OpModVal(
    bEn := TRUE,
    nSel := eOpMode,
    nEn01 := E_BA_AC_OpMod01.eOff,
    bVal01 := arrOpModVal[E_BA_AC_OpMod01.eOff],
    nEn02 := E_BA_AC_OpMod01.eOn,
    bVal02 := arrOpModVal[E_BA_AC_OpMod01.eOn],
    nEn03 := E_BA_AC_OpMod01.eEmergency,
    bVal03 := arrOpModVal[E_BA_AC_OpMod01.eEmergency],
    nEn04 := E_BA_AC_OpMod01.eFrost,
    bVal04 := arrOpModVal[E_BA_AC_OpMod01.eFrost],
    nEn05 := E_BA_AC_OpMod01.eSmokeExtractionProgram,
    bVal05 := arrOpModVal[E_BA_AC_OpMod01.eSmokeExtractionProgram],
    nEn06 := E_BA_AC_OpMod01.eSmokeExtractionSupplyAir,
    bVal06 := arrOpModVal[E_BA_AC_OpMod01.eSmokeExtractionSupplyAir],
    nEn07 := E_BA_AC_OpMod01.eSmokeExtractionExhaustAir,
    bVal07 := arrOpModVal[E_BA_AC_OpMod01.eSmokeExtractionExhaustAir],
    nEn08 := E_BA_AC_OpMod01.eFire,
    bVal08 := arrOpModVal[E_BA_AC_OpMod01.eFire],
    nEn09 := E_BA_AC_OpMod01.eNightCooling,
    bVal09 := arrOpModVal[E_BA_AC_OpMod01.eNightCooling],
    nEn10 := E_BA_AC_OpMod01.eCoolDownProtection,
    bVal10 := arrOpModVal[E_BA_AC_OpMod01.eCoolDownProtection],
    nEn11 := E_BA_AC_OpMod01.eOverHeatingProtection,
    bVal11 := arrOpModVal[E_BA_AC_OpMod01.eOverHeatingProtection],
    nEn12 := E_BA_AC_OpMod01.eAlarm,
    bVal12 := arrOpModVal[E_BA_AC_OpMod01.eAlarm],
    nEn13 := E_BA_AC_OpMod01.eForcedVentilation,
    bVal13 := arrOpModVal[E_BA_AC_OpMod01.eForcedVentilation],
    nEn14 := E_BA_AC_OpMod01.eCentralSwitchOff,
    bVal14 := arrOpModVal[E_BA_AC_OpMod01.eCentralSwitchOff],
    nEn15 := E_BA_AC_OpMod01.eCustomer01,
    bVal15 := arrOpModVal[E_BA_AC_OpMod01.eCustomer01],
    nEn16 := E_BA_AC_OpMod01.eCustomer02,
    bVal16 := arrOpModVal[E_BA_AC_OpMod01.eCustomer02],
    bReplVal := FALSE); // FB_BA_MMUX_B16
bVal := OpModVal.bVal;
_w1 := TO_UDINT(MAX(fDlyOn, 0));
DelayOn(
    bEn := TRUE,
    nSel := eOpMode,
    nEn01 := E_BA_AC_OpMod01.eOff,
    bVal01 := arrIgnoreDelayOnVal[E_BA_AC_OpMod01.eOff],
    nEn02 := E_BA_AC_OpMod01.eOn,
    bVal02 := arrIgnoreDelayOnVal[E_BA_AC_OpMod01.eOn],
    nEn03 := E_BA_AC_OpMod01.eEmergency,
    bVal03 := arrIgnoreDelayOnVal[E_BA_AC_OpMod01.eEmergency],
    nEn04 := E_BA_AC_OpMod01.eFrost,
    bVal04 := arrIgnoreDelayOnVal[E_BA_AC_OpMod01.eFrost],
    nEn05 := E_BA_AC_OpMod01.eSmokeExtractionProgram,
    bVal05 := arrIgnoreDelayOnVal[E_BA_AC_OpMod01.eSmokeExtractionProgram],
    nEn06 := E_BA_AC_OpMod01.eSmokeExtractionSupplyAir,
    bVal06 := arrIgnoreDelayOnVal[E_BA_AC_OpMod01.eSmokeExtractionSupplyAir],
    nEn07 := E_BA_AC_OpMod01.eSmokeExtractionExhaustAir,
    bVal07 := arrIgnoreDelayOnVal[E_BA_AC_OpMod01.eSmokeExtractionExhaustAir],
    nEn08 := E_BA_AC_OpMod01.eFire,
    bVal08 := arrIgnoreDelayOnVal[E_BA_AC_OpMod01.eFire],
    nEn09 := E_BA_AC_OpMod01.eNightCooling,
    bVal09 := arrIgnoreDelayOnVal[E_BA_AC_OpMod01.eNightCooling],
    nEn10 := E_BA_AC_OpMod01.eCoolDownProtection,
    bVal10 := arrIgnoreDelayOnVal[E_BA_AC_OpMod01.eCoolDownProtection],
    nEn11 := E_BA_AC_OpMod01.eOverHeatingProtection,
    bVal11 := arrIgnoreDelayOnVal[E_BA_AC_OpMod01.eOverHeatingProtection],
    nEn12 := E_BA_AC_OpMod01.eAlarm,
    bVal12 := arrIgnoreDelayOnVal[E_BA_AC_OpMod01.eAlarm],
    nEn13 := E_BA_AC_OpMod01.eForcedVentilation,
    bVal13 := arrIgnoreDelayOnVal[E_BA_AC_OpMod01.eForcedVentilation],
    nEn14 := E_BA_AC_OpMod01.eCentralSwitchOff,
    bVal14 := arrIgnoreDelayOnVal[E_BA_AC_OpMod01.eCentralSwitchOff],
    nEn15 := E_BA_AC_OpMod01.eCustomer01,
    bVal15 := arrIgnoreDelayOnVal[E_BA_AC_OpMod01.eCustomer01],
    nEn16 := E_BA_AC_OpMod01.eCustomer02,
    bVal16 := arrIgnoreDelayOnVal[E_BA_AC_OpMod01.eCustomer02],
    bReplVal := FALSE); // FB_BA_MMUX_B16
nDelayOn := SEL(DelayOn.bVal, _w1, 0);
_w2 := TO_UDINT(MAX(fDlyOff, 0));
DelayOff(
    bEn := TRUE,
    nSel := eOpMode,
    nEn01 := E_BA_AC_OpMod01.eOff,
    bVal01 := arrIgnoreDelayOffVal[E_BA_AC_OpMod01.eOff],
    nEn02 := E_BA_AC_OpMod01.eOn,
    bVal02 := arrIgnoreDelayOffVal[E_BA_AC_OpMod01.eOn],
    nEn03 := E_BA_AC_OpMod01.eEmergency,
    bVal03 := arrIgnoreDelayOffVal[E_BA_AC_OpMod01.eEmergency],
    nEn04 := E_BA_AC_OpMod01.eFrost,
    bVal04 := arrIgnoreDelayOffVal[E_BA_AC_OpMod01.eFrost],
    nEn05 := E_BA_AC_OpMod01.eSmokeExtractionProgram,
    bVal05 := arrIgnoreDelayOffVal[E_BA_AC_OpMod01.eSmokeExtractionProgram],
    nEn06 := E_BA_AC_OpMod01.eSmokeExtractionSupplyAir,
    bVal06 := arrIgnoreDelayOffVal[E_BA_AC_OpMod01.eSmokeExtractionSupplyAir],
    nEn07 := E_BA_AC_OpMod01.eSmokeExtractionExhaustAir,
    bVal07 := arrIgnoreDelayOffVal[E_BA_AC_OpMod01.eSmokeExtractionExhaustAir],
    nEn08 := E_BA_AC_OpMod01.eFire,
    bVal08 := arrIgnoreDelayOffVal[E_BA_AC_OpMod01.eFire],
    nEn09 := E_BA_AC_OpMod01.eNightCooling,
    bVal09 := arrIgnoreDelayOffVal[E_BA_AC_OpMod01.eNightCooling],
    nEn10 := E_BA_AC_OpMod01.eCoolDownProtection,
    bVal10 := arrIgnoreDelayOffVal[E_BA_AC_OpMod01.eCoolDownProtection],
    nEn11 := E_BA_AC_OpMod01.eOverHeatingProtection,
    bVal11 := arrIgnoreDelayOffVal[E_BA_AC_OpMod01.eOverHeatingProtection],
    nEn12 := E_BA_AC_OpMod01.eAlarm,
    bVal12 := arrIgnoreDelayOffVal[E_BA_AC_OpMod01.eAlarm],
    nEn13 := E_BA_AC_OpMod01.eForcedVentilation,
    bVal13 := arrIgnoreDelayOffVal[E_BA_AC_OpMod01.eForcedVentilation],
    nEn14 := E_BA_AC_OpMod01.eCentralSwitchOff,
    bVal14 := arrIgnoreDelayOffVal[E_BA_AC_OpMod01.eCentralSwitchOff],
    nEn15 := E_BA_AC_OpMod01.eCustomer01,
    bVal15 := arrIgnoreDelayOffVal[E_BA_AC_OpMod01.eCustomer01],
    nEn16 := E_BA_AC_OpMod01.eCustomer02,
    bVal16 := arrIgnoreDelayOffVal[E_BA_AC_OpMod01.eCustomer02],
    bReplVal := FALSE); // FB_BA_MMUX_B16
nDelayOff := SEL(DelayOff.bVal, _w2, 0);
IgnoreFdb(
    bEn := TRUE,
    nSel := eOpMode,
    nEn01 := E_BA_AC_OpMod01.eOff,
    bVal01 := arrIgnoreFdbVal[E_BA_AC_OpMod01.eOff],
    nEn02 := E_BA_AC_OpMod01.eOn,
    bVal02 := arrIgnoreFdbVal[E_BA_AC_OpMod01.eOn],
    nEn03 := E_BA_AC_OpMod01.eEmergency,
    bVal03 := arrIgnoreFdbVal[E_BA_AC_OpMod01.eEmergency],
    nEn04 := E_BA_AC_OpMod01.eFrost,
    bVal04 := arrIgnoreFdbVal[E_BA_AC_OpMod01.eFrost],
    nEn05 := E_BA_AC_OpMod01.eSmokeExtractionProgram,
    bVal05 := arrIgnoreFdbVal[E_BA_AC_OpMod01.eSmokeExtractionProgram],
    nEn06 := E_BA_AC_OpMod01.eSmokeExtractionSupplyAir,
    bVal06 := arrIgnoreFdbVal[E_BA_AC_OpMod01.eSmokeExtractionSupplyAir],
    nEn07 := E_BA_AC_OpMod01.eSmokeExtractionExhaustAir,
    bVal07 := arrIgnoreFdbVal[E_BA_AC_OpMod01.eSmokeExtractionExhaustAir],
    nEn08 := E_BA_AC_OpMod01.eFire,
    bVal08 := arrIgnoreFdbVal[E_BA_AC_OpMod01.eFire],
    nEn09 := E_BA_AC_OpMod01.eNightCooling,
    bVal09 := arrIgnoreFdbVal[E_BA_AC_OpMod01.eNightCooling],
    nEn10 := E_BA_AC_OpMod01.eCoolDownProtection,
    bVal10 := arrIgnoreFdbVal[E_BA_AC_OpMod01.eCoolDownProtection],
    nEn11 := E_BA_AC_OpMod01.eOverHeatingProtection,
    bVal11 := arrIgnoreFdbVal[E_BA_AC_OpMod01.eOverHeatingProtection],
    nEn12 := E_BA_AC_OpMod01.eAlarm,
    bVal12 := arrIgnoreFdbVal[E_BA_AC_OpMod01.eAlarm],
    nEn13 := E_BA_AC_OpMod01.eForcedVentilation,
    bVal13 := arrIgnoreFdbVal[E_BA_AC_OpMod01.eForcedVentilation],
    nEn14 := E_BA_AC_OpMod01.eCentralSwitchOff,
    bVal14 := arrIgnoreFdbVal[E_BA_AC_OpMod01.eCentralSwitchOff],
    nEn15 := E_BA_AC_OpMod01.eCustomer01,
    bVal15 := arrIgnoreFdbVal[E_BA_AC_OpMod01.eCustomer01],
    nEn16 := E_BA_AC_OpMod01.eCustomer02,
    bVal16 := arrIgnoreFdbVal[E_BA_AC_OpMod01.eCustomer02],
    bReplVal := FALSE); // FB_BA_MMUX_B16
_bFdb := SEL(IgnoreFdb.bVal, bFdb, TRUE);

END_FUNCTION_BLOCK

// ---- Templates/POUs/Trade/AirConditioning/General/FB_BA_AC_OpModAggMdlt.TcPOU
{region '#Template'}
	{attribute 'Version' := '5.1.0.0'}
	{attribute 'Tags' := '"LCID": "1031", "Text": "AC, Allgemein, AHU, Betriebsart"'}
	{attribute 'Tags' := '"LCID": "1033", "Text": "AC, General, AHU, Operating mode"'}
	{attribute 'Using' := '"Type": "Template", "URI": "E_BA_AC_OpMod01"'}
	{attribute 'Description' := '"LCID": "1031", "Text": "Betriebsart"'}
	{attribute 'Description' := '"LCID": "1033", "Text": "Operating mode"'}
{endregion}

FUNCTION_BLOCK FB_BA_AC_OpModAggMdlt
VAR_INPUT
	stPriorityEn				: ST_BA_PriorityEn;	
	eOpMode					: E_BA_AC_OpMod01;
	bFdb					: BOOL;
	fDlyOn					: REAL;	
	fDlyOff					: REAL;	
END_VAR
VAR_OUTPUT
	stCmd					: ST_BA_Mdlt;
	nRemSecStepUp           : UDINT;
	nRemSecStepDown         : UDINT;
END_VAR
VAR_IN_OUT
	stStep					: ST_BA_Step;
END_VAR
VAR_INPUT CONSTANT
	OpModVal				: FB_BA_MMUX_UDI16;
	DelayOn					: FB_BA_MMUX_B16;
	DelayOff				: FB_BA_MMUX_B16;
	IgnoreFdb				: FB_BA_MMUX_B16;	
	Step                    : FB_BA_StepMdlt;
END_VAR
VAR_INPUT CONSTANT PERSISTENT
	bInit					: BOOL := TRUE;
	arrOpModVal				: ARRAY [1..16] OF E_BA_Mdlt;
	arrIgnoreDelayOnVal 	: ARRAY [1..16] OF BOOL;
	arrIgnoreDelayOffVal	: ARRAY [1..16] OF BOOL;
	arrIgnoreFdbVal 		: ARRAY [1..16] OF BOOL;	
END_VAR
VAR
	eVal					: E_BA_Mdlt;
	_bFdb					: BOOL;	
	nDelayOn				: UDINT;
	nDelayOff				: UDINT;	
END_VAR
VAR // added by the converter: edge detectors and wires of the graphical bodies
    _w1, _w2 : UDINT;
END_VAR

OpModVal(
    bEn := TRUE,
    nSel := eOpMode,
    nEn01 := E_BA_AC_OpMod01.eOff,
    nVal01 := arrOpModVal[E_BA_AC_OpMod01.eOff],
    nEn02 := E_BA_AC_OpMod01.eOn,
    nVal02 := arrOpModVal[E_BA_AC_OpMod01.eOn],
    nEn03 := E_BA_AC_OpMod01.eEmergency,
    nVal03 := arrOpModVal[E_BA_AC_OpMod01.eEmergency],
    nEn04 := E_BA_AC_OpMod01.eFrost,
    nVal04 := arrOpModVal[E_BA_AC_OpMod01.eFrost],
    nEn05 := E_BA_AC_OpMod01.eSmokeExtractionProgram,
    nVal05 := arrOpModVal[E_BA_AC_OpMod01.eSmokeExtractionProgram],
    nEn06 := E_BA_AC_OpMod01.eSmokeExtractionSupplyAir,
    nVal06 := arrOpModVal[E_BA_AC_OpMod01.eSmokeExtractionSupplyAir],
    nEn07 := E_BA_AC_OpMod01.eSmokeExtractionExhaustAir,
    nVal07 := arrOpModVal[E_BA_AC_OpMod01.eSmokeExtractionExhaustAir],
    nEn08 := E_BA_AC_OpMod01.eFire,
    nVal08 := arrOpModVal[E_BA_AC_OpMod01.eFire],
    nEn09 := E_BA_AC_OpMod01.eNightCooling,
    nVal09 := arrOpModVal[E_BA_AC_OpMod01.eNightCooling],
    nEn10 := E_BA_AC_OpMod01.eCoolDownProtection,
    nVal10 := arrOpModVal[E_BA_AC_OpMod01.eCoolDownProtection],
    nEn11 := E_BA_AC_OpMod01.eOverHeatingProtection,
    nVal11 := arrOpModVal[E_BA_AC_OpMod01.eOverHeatingProtection],
    nEn12 := E_BA_AC_OpMod01.eAlarm,
    nVal12 := arrOpModVal[E_BA_AC_OpMod01.eAlarm],
    nEn13 := E_BA_AC_OpMod01.eForcedVentilation,
    nVal13 := arrOpModVal[E_BA_AC_OpMod01.eForcedVentilation],
    nEn14 := E_BA_AC_OpMod01.eCentralSwitchOff,
    nVal14 := arrOpModVal[E_BA_AC_OpMod01.eCentralSwitchOff],
    nEn15 := E_BA_AC_OpMod01.eCustomer01,
    nVal15 := arrOpModVal[E_BA_AC_OpMod01.eCustomer01],
    nEn16 := E_BA_AC_OpMod01.eCustomer02,
    nVal16 := arrOpModVal[E_BA_AC_OpMod01.eCustomer02],
    nReplVal := E_BA_Mdlt.eOff); // FB_BA_MMUX_UDI16
eVal := OpModVal.nVal;
_w1 := TO_UDINT(MAX(fDlyOn, 0));
DelayOn(
    bEn := TRUE,
    nSel := eOpMode,
    nEn01 := E_BA_AC_OpMod01.eOff,
    bVal01 := arrIgnoreDelayOnVal[E_BA_AC_OpMod01.eOff],
    nEn02 := E_BA_AC_OpMod01.eOn,
    bVal02 := arrIgnoreDelayOnVal[E_BA_AC_OpMod01.eOn],
    nEn03 := E_BA_AC_OpMod01.eEmergency,
    bVal03 := arrIgnoreDelayOnVal[E_BA_AC_OpMod01.eEmergency],
    nEn04 := E_BA_AC_OpMod01.eFrost,
    bVal04 := arrIgnoreDelayOnVal[E_BA_AC_OpMod01.eFrost],
    nEn05 := E_BA_AC_OpMod01.eSmokeExtractionProgram,
    bVal05 := arrIgnoreDelayOnVal[E_BA_AC_OpMod01.eSmokeExtractionProgram],
    nEn06 := E_BA_AC_OpMod01.eSmokeExtractionSupplyAir,
    bVal06 := arrIgnoreDelayOnVal[E_BA_AC_OpMod01.eSmokeExtractionSupplyAir],
    nEn07 := E_BA_AC_OpMod01.eSmokeExtractionExhaustAir,
    bVal07 := arrIgnoreDelayOnVal[E_BA_AC_OpMod01.eSmokeExtractionExhaustAir],
    nEn08 := E_BA_AC_OpMod01.eFire,
    bVal08 := arrIgnoreDelayOnVal[E_BA_AC_OpMod01.eFire],
    nEn09 := E_BA_AC_OpMod01.eNightCooling,
    bVal09 := arrIgnoreDelayOnVal[E_BA_AC_OpMod01.eNightCooling],
    nEn10 := E_BA_AC_OpMod01.eCoolDownProtection,
    bVal10 := arrIgnoreDelayOnVal[E_BA_AC_OpMod01.eCoolDownProtection],
    nEn11 := E_BA_AC_OpMod01.eOverHeatingProtection,
    bVal11 := arrIgnoreDelayOnVal[E_BA_AC_OpMod01.eOverHeatingProtection],
    nEn12 := E_BA_AC_OpMod01.eAlarm,
    bVal12 := arrIgnoreDelayOnVal[E_BA_AC_OpMod01.eAlarm],
    nEn13 := E_BA_AC_OpMod01.eForcedVentilation,
    bVal13 := arrIgnoreDelayOnVal[E_BA_AC_OpMod01.eForcedVentilation],
    nEn14 := E_BA_AC_OpMod01.eCentralSwitchOff,
    bVal14 := arrIgnoreDelayOnVal[E_BA_AC_OpMod01.eCentralSwitchOff],
    nEn15 := E_BA_AC_OpMod01.eCustomer01,
    bVal15 := arrIgnoreDelayOnVal[E_BA_AC_OpMod01.eCustomer01],
    nEn16 := E_BA_AC_OpMod01.eCustomer02,
    bVal16 := arrIgnoreDelayOnVal[E_BA_AC_OpMod01.eCustomer02],
    bReplVal := FALSE); // FB_BA_MMUX_B16
nDelayOn := SEL(DelayOn.bVal, _w1, 0);
_w2 := TO_UDINT(MAX(fDlyOff, 0));
DelayOff(
    bEn := TRUE,
    nSel := eOpMode,
    nEn01 := E_BA_AC_OpMod01.eOff,
    bVal01 := arrIgnoreDelayOffVal[E_BA_AC_OpMod01.eOff],
    nEn02 := E_BA_AC_OpMod01.eOn,
    bVal02 := arrIgnoreDelayOffVal[E_BA_AC_OpMod01.eOn],
    nEn03 := E_BA_AC_OpMod01.eEmergency,
    bVal03 := arrIgnoreDelayOffVal[E_BA_AC_OpMod01.eEmergency],
    nEn04 := E_BA_AC_OpMod01.eFrost,
    bVal04 := arrIgnoreDelayOffVal[E_BA_AC_OpMod01.eFrost],
    nEn05 := E_BA_AC_OpMod01.eSmokeExtractionProgram,
    bVal05 := arrIgnoreDelayOffVal[E_BA_AC_OpMod01.eSmokeExtractionProgram],
    nEn06 := E_BA_AC_OpMod01.eSmokeExtractionSupplyAir,
    bVal06 := arrIgnoreDelayOffVal[E_BA_AC_OpMod01.eSmokeExtractionSupplyAir],
    nEn07 := E_BA_AC_OpMod01.eSmokeExtractionExhaustAir,
    bVal07 := arrIgnoreDelayOffVal[E_BA_AC_OpMod01.eSmokeExtractionExhaustAir],
    nEn08 := E_BA_AC_OpMod01.eFire,
    bVal08 := arrIgnoreDelayOffVal[E_BA_AC_OpMod01.eFire],
    nEn09 := E_BA_AC_OpMod01.eNightCooling,
    bVal09 := arrIgnoreDelayOffVal[E_BA_AC_OpMod01.eNightCooling],
    nEn10 := E_BA_AC_OpMod01.eCoolDownProtection,
    bVal10 := arrIgnoreDelayOffVal[E_BA_AC_OpMod01.eCoolDownProtection],
    nEn11 := E_BA_AC_OpMod01.eOverHeatingProtection,
    bVal11 := arrIgnoreDelayOffVal[E_BA_AC_OpMod01.eOverHeatingProtection],
    nEn12 := E_BA_AC_OpMod01.eAlarm,
    bVal12 := arrIgnoreDelayOffVal[E_BA_AC_OpMod01.eAlarm],
    nEn13 := E_BA_AC_OpMod01.eForcedVentilation,
    bVal13 := arrIgnoreDelayOffVal[E_BA_AC_OpMod01.eForcedVentilation],
    nEn14 := E_BA_AC_OpMod01.eCentralSwitchOff,
    bVal14 := arrIgnoreDelayOffVal[E_BA_AC_OpMod01.eCentralSwitchOff],
    nEn15 := E_BA_AC_OpMod01.eCustomer01,
    bVal15 := arrIgnoreDelayOffVal[E_BA_AC_OpMod01.eCustomer01],
    nEn16 := E_BA_AC_OpMod01.eCustomer02,
    bVal16 := arrIgnoreDelayOffVal[E_BA_AC_OpMod01.eCustomer02],
    bReplVal := FALSE); // FB_BA_MMUX_B16
nDelayOff := SEL(DelayOff.bVal, _w2, 0);
IgnoreFdb(
    bEn := TRUE,
    nSel := eOpMode,
    nEn01 := E_BA_AC_OpMod01.eOff,
    bVal01 := arrIgnoreFdbVal[E_BA_AC_OpMod01.eOff],
    nEn02 := E_BA_AC_OpMod01.eOn,
    bVal02 := arrIgnoreFdbVal[E_BA_AC_OpMod01.eOn],
    nEn03 := E_BA_AC_OpMod01.eEmergency,
    bVal03 := arrIgnoreFdbVal[E_BA_AC_OpMod01.eEmergency],
    nEn04 := E_BA_AC_OpMod01.eFrost,
    bVal04 := arrIgnoreFdbVal[E_BA_AC_OpMod01.eFrost],
    nEn05 := E_BA_AC_OpMod01.eSmokeExtractionProgram,
    bVal05 := arrIgnoreFdbVal[E_BA_AC_OpMod01.eSmokeExtractionProgram],
    nEn06 := E_BA_AC_OpMod01.eSmokeExtractionSupplyAir,
    bVal06 := arrIgnoreFdbVal[E_BA_AC_OpMod01.eSmokeExtractionSupplyAir],
    nEn07 := E_BA_AC_OpMod01.eSmokeExtractionExhaustAir,
    bVal07 := arrIgnoreFdbVal[E_BA_AC_OpMod01.eSmokeExtractionExhaustAir],
    nEn08 := E_BA_AC_OpMod01.eFire,
    bVal08 := arrIgnoreFdbVal[E_BA_AC_OpMod01.eFire],
    nEn09 := E_BA_AC_OpMod01.eNightCooling,
    bVal09 := arrIgnoreFdbVal[E_BA_AC_OpMod01.eNightCooling],
    nEn10 := E_BA_AC_OpMod01.eCoolDownProtection,
    bVal10 := arrIgnoreFdbVal[E_BA_AC_OpMod01.eCoolDownProtection],
    nEn11 := E_BA_AC_OpMod01.eOverHeatingProtection,
    bVal11 := arrIgnoreFdbVal[E_BA_AC_OpMod01.eOverHeatingProtection],
    nEn12 := E_BA_AC_OpMod01.eAlarm,
    bVal12 := arrIgnoreFdbVal[E_BA_AC_OpMod01.eAlarm],
    nEn13 := E_BA_AC_OpMod01.eForcedVentilation,
    bVal13 := arrIgnoreFdbVal[E_BA_AC_OpMod01.eForcedVentilation],
    nEn14 := E_BA_AC_OpMod01.eCentralSwitchOff,
    bVal14 := arrIgnoreFdbVal[E_BA_AC_OpMod01.eCentralSwitchOff],
    nEn15 := E_BA_AC_OpMod01.eCustomer01,
    bVal15 := arrIgnoreFdbVal[E_BA_AC_OpMod01.eCustomer01],
    nEn16 := E_BA_AC_OpMod01.eCustomer02,
    bVal16 := arrIgnoreFdbVal[E_BA_AC_OpMod01.eCustomer02],
    bReplVal := FALSE); // FB_BA_MMUX_B16
_bFdb := SEL(IgnoreFdb.bVal, bFdb, TRUE);
Step(
    stPriorityEn := stPriorityEn,
    eVal := eVal,
    bFdb := _bFdb,
    nDlyOn := nDelayOn,
    nDlyOff := nDelayOff,
    stStep := stStep); // FB_BA_StepMdlt
stCmd := Step.stCmd;
nRemSecStepUp := Step.nRemSecStepUp;
nRemSecStepDown := Step.nRemSecStepDown;

END_FUNCTION_BLOCK

// ---- Templates/POUs/Trade/AirConditioning/General/FB_BA_AC_PlantCmd_AHU_1st_10.TcPOU
{region '#Template'}
	{attribute 'Version' := '5.1.0.0'}
	{attribute 'Tags' := '"LCID": "1031", "Text": "AC, Allgemein, AHU, Startprogramm, Aggregat, Kommandierung"'}
	{attribute 'Tags' := '"LCID": "1033", "Text": "AC, General, AHU, Start program, Aggregate, Command"'}
	{attribute 'Using' := '"Type": "Template", "URI": "E_BA_AC_PlantStep01"'}
	{attribute 'Using' := '"Type": "Template", "URI": "E_BA_AC_OpMod01"'}
	{attribute 'Description' := '"LCID": "1031", "Text": "Kommandierung der Anlage FB_BA_AHU_1st_10"'}
	{attribute 'Description' := '"LCID": "1033", "Text": "Commanding the plant FB_BA_AHU_1st_10"'}
{endregion}

FUNCTION_BLOCK FB_BA_AC_PlantCmd_AHU_1st_10 EXTENDS FB_BA_View
VAR_INPUT
	eOpMode						: E_BA_AC_OpMod01;
	stPriorityEn				: ST_BA_PriorityEn;	
	bDmpOuAOpn					: BOOL;		//	Rückmeldung Aussenluftklappe offen		//	Feedback outside air damper open
	bDmpExhAOpn					: BOOL;		//	Rückmeldung Fortluftklappe offen		//	Feedback exhaust air damper open
	bPreRinse					: BOOL;		//	Vorspülen abgeschlossen					//	Prerinse ready
END_VAR
VAR_OUTPUT
	ePltStp						: E_BA_AC_PlantStep01;	//	Stufen des Anlagenstarts	//	Stages of the plant starts	
	stOuADmp					: ST_BA_Binary;
	stExhADmp					: ST_BA_Binary;
	stSuAFan					: ST_BA_Mdlt;
	stExtAFan					: ST_BA_Mdlt;
	stPreHtr					: ST_BA_Binary;
	stCooler					: ST_BA_Binary;
	stErc						: ST_BA_Binary;
	stTempCtrl					: ST_BA_Mdlt;
	bStepCtrlUp					: BOOL;
	bStepCtrlDown				: BOOL;	
END_VAR
VAR_INPUT CONSTANT
	DmpDlyCls					: FB_BA_AV_Op;
	SuAFanDlyOn					: FB_BA_AV_Op;
	ExtAFanDlyOn				: FB_BA_AV_Op;
	TempCtrlDlyOn				: FB_BA_AV_Op;
	PltStp						: FB_BA_MV_Op;
	
	StepCtrlAgg					: FB_BA_StepCtrlAgg16; //	Schrittsteuerung Aggregate // Step control aggregate	
	
	ErcOpMod					: FB_BA_AC_OpModAggBinary;
	PreHtrOpMod					: FB_BA_AC_OpModAggBinary;
	OuADmpOpMod					: FB_BA_AC_OpModAggBinary;
	SuAFanOpMod					: FB_BA_AC_OpModAggMdlt;
	ExhADmpOpMod				: FB_BA_AC_OpModAggBinary;
	ExtAFanOpMod				: FB_BA_AC_OpModAggMdlt;
	CoolerOpMod					: FB_BA_AC_OpModAggBinary;
	TempCtrlOpMod				: FB_BA_AC_OpModAggMdlt;
END_VAR
VAR
	stAgg01						: ST_BA_Step;
	stAgg02						: ST_BA_Step;
	stAgg03						: ST_BA_Step;
	stAgg04						: ST_BA_Step;
	stAgg05						: ST_BA_Step;
	stAgg06						: ST_BA_Step;
	stAgg07						: ST_BA_Step;
	stAgg08						: ST_BA_Step;
	stAgg09						: ST_BA_Step;
	stAgg10						: ST_BA_Step;
	stAgg11						: ST_BA_Step;
	stAgg12						: ST_BA_Step;	
	stAgg13						: ST_BA_Step;	
	stAgg14						: ST_BA_Step;	
	stAgg15						: ST_BA_Step;	
	stAgg16						: ST_BA_Step;	
	
	PltStpMMUX					: FB_BA_MMUX_UDI16;	//	Stufen des Anlagenstarts	//	Stages of the plant starts	
END_VAR

SUPER^(); // FB_BA_View
CallInit();
DmpDlyCls(); // FB_BA_AV_Op
TempCtrlDlyOn(); // FB_BA_AV_Op
SuAFanDlyOn(); // FB_BA_AV_Op
ExtAFanDlyOn(); // FB_BA_AV_Op
StepCtrlAgg(
    bEnUpDown := stPriorityEn.bPlt,
    nNumOfAgg := 8,
    stAgg01 := stAgg01,
    stAgg02 := stAgg02,
    stAgg03 := stAgg03,
    stAgg04 := stAgg04,
    stAgg05 := stAgg05,
    stAgg06 := stAgg06,
    stAgg07 := stAgg07,
    stAgg08 := stAgg08,
    stAgg09 := stAgg09,
    stAgg10 := stAgg10,
    stAgg11 := stAgg11,
    stAgg12 := stAgg12,
    stAgg13 := stAgg13,
    stAgg14 := stAgg14,
    stAgg15 := stAgg15,
    stAgg16 := stAgg16); // FB_BA_StepCtrlAgg16
bStepCtrlUp := StepCtrlAgg.bUp;
bStepCtrlDown := StepCtrlAgg.bDown;
PltStpMMUX(
    bEn := TRUE,
    nSel := StepCtrlAgg.nStep + 1,
    nEn01 := 16,
    nEn02 := 15,
    nEn03 := 14,
    nEn04 := 13,
    nEn05 := 12,
    nEn06 := 11,
    nEn07 := 10,
    nVal07 := E_BA_AC_PlantStep01.eOn,
    nEn08 := 9,
    nVal08 := E_BA_AC_PlantStep01.eEnablingTemperatureControl,
    nEn09 := 8,
    nVal09 := E_BA_AC_PlantStep01.eCooler,
    nEn10 := 7,
    nVal10 := E_BA_AC_PlantStep01.eFanExtractAir,
    nEn11 := 6,
    nVal11 := E_BA_AC_PlantStep01.eDamperExhA,
    nEn12 := 5,
    nVal12 := E_BA_AC_PlantStep01.eFanSupplyAir,
    nEn13 := 4,
    nVal13 := E_BA_AC_PlantStep01.eDamperOuA,
    nEn14 := 3,
    nVal14 := E_BA_AC_PlantStep01.ePreRinse,
    nEn15 := 2,
    nVal15 := E_BA_AC_PlantStep01.eErc,
    nEn16 := 1,
    nVal16 := E_BA_AC_PlantStep01.eOff); // FB_BA_MMUX_UDI16
PltStp(nValuePgm := PltStpMMUX.nVal); // FB_BA_MV_Op
ePltStp := PltStp.nPresentValue;
ErcOpMod(stPriorityEn := stPriorityEn, eOpMode := eOpMode, stStep := stAgg01); // FB_BA_AC_OpModAggBinary
stErc := ErcOpMod.stCmd;
PreHtrOpMod(stPriorityEn := stPriorityEn, eOpMode := eOpMode, bFdb := bPreRinse, stStep := stAgg02); // FB_BA_AC_OpModAggBinary
stPreHtr := PreHtrOpMod.stCmd;
OuADmpOpMod(
    stPriorityEn := stPriorityEn,
    eOpMode := eOpMode,
    bFdb := bDmpOuAOpn,
    fDlyOn := SuAFanDlyOn.fPresentValue,
    fDlyOff := DmpDlyCls.fPresentValue,
    stStep := stAgg03); // FB_BA_AC_OpModAggBinary
stOuADmp := OuADmpOpMod.stCmd;
SuAFanOpMod(stPriorityEn := stPriorityEn, eOpMode := eOpMode, stStep := stAgg04); // FB_BA_AC_OpModAggMdlt
stSuAFan := SuAFanOpMod.stCmd;
ExhADmpOpMod(
    stPriorityEn := stPriorityEn,
    eOpMode := eOpMode,
    bFdb := bDmpExhAOpn,
    fDlyOn := ExtAFanDlyOn.fPresentValue,
    fDlyOff := DmpDlyCls.fPresentValue,
    stStep := stAgg05); // FB_BA_AC_OpModAggBinary
stExhADmp := ExhADmpOpMod.stCmd;
ExtAFanOpMod(stPriorityEn := stPriorityEn, eOpMode := eOpMode, stStep := stAgg06); // FB_BA_AC_OpModAggMdlt
stExtAFan := ExtAFanOpMod.stCmd;
CoolerOpMod(stPriorityEn := stPriorityEn, eOpMode := eOpMode, stStep := stAgg07); // FB_BA_AC_OpModAggBinary
stCooler := CoolerOpMod.stCmd;
TempCtrlOpMod(
    stPriorityEn := stPriorityEn,
    eOpMode := eOpMode,
    fDlyOn := TempCtrlDlyOn.fPresentValue,
    stStep := stAgg08); // FB_BA_AC_OpModAggMdlt
stTempCtrl := TempCtrlOpMod.stCmd;

METHOD CallInit
VAR_INPUT
END_VAR
InitErc();
InitPreHtr();

InitOuADmp();
InitSuAFan();

InitExhADmp();
InitExtAFan();

InitCooler();

InitTempCtrl();
END_METHOD

METHOD FB_init : BOOL
VAR_INPUT
	bInitRetains : BOOL; // if TRUE, the retain variables are initialized (warm start / cold start)
	bInCopyCode : BOOL;  // if TRUE, the instance afterwards gets moved into the copy code (online change)
END_VAR
DmpDlyCls.iParent			:= THIS^;
DmpDlyCls.iLabel			:= LblCtl_TimeDelayDampersClose; 	
DmpDlyCls.eUnit				:= E_BA_Unit.eTime_Seconds;  
DmpDlyCls.fValueRm			:= 10;

SuAFanDlyOn.iParent			:= THIS^;
SuAFanDlyOn.iLabel			:= LblCtl_TimeDelaySupplyAirFanOn;   		
SuAFanDlyOn.eUnit			:= E_BA_Unit.eTime_Seconds;  
SuAFanDlyOn.fValueRm		:= 10;

ExtAFanDlyOn.iParent		:= THIS^;
ExtAFanDlyOn.iLabel			:= LblCtl_TimeDelayExtractAirFanOn;   	
ExtAFanDlyOn.eUnit			:= E_BA_Unit.eTime_Seconds;  
ExtAFanDlyOn.fValueRm		:= 10;

TempCtrlDlyOn.iParent		:= THIS^;
TempCtrlDlyOn.iLabel		:= LblCtl_TimeDelayTemperatureSequenceControlOn;   	
TempCtrlDlyOn.eUnit			:= E_BA_Unit.eTime_Seconds;  
TempCtrlDlyOn.fValueRm		:= 5;

PltStp.iParent				:= THIS^;
PltStp.iLabel				:= LblCtl_StagesOfThePlantStartup; 	
PltStp.aStateText[1]		:= txtEvent_Off;
PltStp.aStateText[2]		:= txtEvent_EnergyRecovery;
PltStp.aStateText[3]		:= txtEvent_PreRinse;// or txtEvent_Preheater
PltStp.aStateText[4]		:= txtEvent_DamperOutsideAir;
PltStp.aStateText[5]		:= txtEvent_SupplyAirFan;
PltStp.aStateText[6]		:= txtEvent_DamperExhaustAir;
PltStp.aStateText[7]		:= txtEvent_ExtractAirFan;
PltStp.aStateText[8]		:= txtEvent_Cooler;
PltStp.aStateText[9]		:= txtEvent_Reheater;
PltStp.aStateText[10]		:= txtEvent_MixedAir;
PltStp.aStateText[11]		:= txtEvent_EnableTemperatureControl;
PltStp.aStateText[12]		:= txtEvent_EnableHumidityControl;
PltStp.aStateText[13]		:= txtEvent_On;
END_METHOD

METHOD InitCooler
VAR_INPUT
END_VAR
IF	CoolerOpMod.bInit
THEN	
	CoolerOpMod.bInit := FALSE;
	//////////////////////////////////////////////
	//////////////////////////////////////////////
	//	E_BA_AC_OpMod01.eOff
	CoolerOpMod.arrOpModVal[E_BA_AC_OpMod01.eOff]				:= FALSE;
	CoolerOpMod.arrIgnoreDelayOnVal[E_BA_AC_OpMod01.eOff]		:= TRUE;
	CoolerOpMod.arrIgnoreDelayOffVal[E_BA_AC_OpMod01.eOff]		:= TRUE;
	CoolerOpMod.arrIgnoreFdbVal[E_BA_AC_OpMod01.eOff]			:= TRUE;
	//////////////////////////////////////////////
	//////////////////////////////////////////////
	//	E_BA_AC_OpMod01.eOn
	CoolerOpMod.arrOpModVal[E_BA_AC_OpMod01.eOn]				:= TRUE;
	CoolerOpMod.arrIgnoreDelayOnVal[E_BA_AC_OpMod01.eOn]		:= TRUE;
	CoolerOpMod.arrIgnoreDelayOffVal[E_BA_AC_OpMod01.eOn]		:= TRUE;
	CoolerOpMod.arrIgnoreFdbVal[E_BA_AC_OpMod01.eOn]			:= TRUE;
	//////////////////////////////////////////////
	//////////////////////////////////////////////
	//	E_BA_AC_OpMod01.eEmergency
	CoolerOpMod.arrOpModVal[E_BA_AC_OpMod01.eEmergency]				:= FALSE;
	CoolerOpMod.arrIgnoreDelayOnVal[E_BA_AC_OpMod01.eEmergency]		:= TRUE;
	CoolerOpMod.arrIgnoreDelayOffVal[E_BA_AC_OpMod01.eEmergency]	:= TRUE;
	CoolerOpMod.arrIgnoreFdbVal[E_BA_AC_OpMod01.eEmergency]			:= TRUE;
	//////////////////////////////////////////////
	//////////////////////////////////////////////
	//	E_OpModBA_AC_OpMod01.eFrost
	CoolerOpMod.arrOpModVal[E_BA_AC_OpMod01.eFrost]				:= FALSE;
	CoolerOpMod.arrIgnoreDelayOnVal[E_BA_AC_OpMod01.eFrost]		:= TRUE;
	CoolerOpMod.arrIgnoreDelayOffVal[E_BA_AC_OpMod01.eFrost]	:= TRUE;
	CoolerOpMod.arrIgnoreFdbVal[E_BA_AC_OpMod01.eFrost]			:= TRUE;
	//////////////////////////////////////////////
	//////////////////////////////////////////////
	//	E_BA_AC_OpMod01.eSmokeExtractionProgramm
	CoolerOpMod.arrOpModVal[E_BA_AC_OpMod01.eSmokeExtractionProgram]				:= FALSE;
	CoolerOpMod.arrIgnoreDelayOnVal[E_BA_AC_OpMod01.eSmokeExtractionProgram]		:= TRUE;
	CoolerOpMod.arrIgnoreDelayOffVal[E_BA_AC_OpMod01.eSmokeExtractionProgram]		:= TRUE;
	CoolerOpMod.arrIgnoreFdbVal[E_BA_AC_OpMod01.eSmokeExtractionProgram]			:= TRUE;
	//////////////////////////////////////////////
	//////////////////////////////////////////////
	//	E_BA_AC_OpMod01.eSmokeExtractionSupplyAir
	CoolerOpMod.arrOpModVal[E_BA_AC_OpMod01.eSmokeExtractionSupplyAir]				:= FALSE;
	CoolerOpMod.arrIgnoreDelayOnVal[E_BA_AC_OpMod01.eSmokeExtractionSupplyAir]		:= TRUE;
	CoolerOpMod.arrIgnoreDelayOffVal[E_BA_AC_OpMod01.eSmokeExtractionSupplyAir]		:= TRUE;
	CoolerOpMod.arrIgnoreFdbVal[E_BA_AC_OpMod01.eSmokeExtractionSupplyAir]			:= TRUE;
	//////////////////////////////////////////////
	//////////////////////////////////////////////
	//	E_BA_AC_OpMod01.eSmokeExtractionExhaustAir
	CoolerOpMod.arrOpModVal[E_BA_AC_OpMod01.eSmokeExtractionExhaustAir]				:= FALSE;
	CoolerOpMod.arrIgnoreDelayOnVal[E_BA_AC_OpMod01.eSmokeExtractionExhaustAir]		:= TRUE;
	CoolerOpMod.arrIgnoreDelayOffVal[E_BA_AC_OpMod01.eSmokeExtractionExhaustAir]	:= TRUE;
	CoolerOpMod.arrIgnoreFdbVal[E_BA_AC_OpMod01.eSmokeExtractionExhaustAir]			:= TRUE;
	//////////////////////////////////////////////
	//////////////////////////////////////////////
	//	E_BA_AC_OpMod01.eFire
	CoolerOpMod.arrOpModVal[E_BA_AC_OpMod01.eFire]				:= FALSE;
	CoolerOpMod.arrIgnoreDelayOnVal[E_BA_AC_OpMod01.eFire]		:= TRUE;
	CoolerOpMod.arrIgnoreDelayOffVal[E_BA_AC_OpMod01.eFire]		:= TRUE;
	CoolerOpMod.arrIgnoreFdbVal[E_BA_AC_OpMod01.eFire]			:= TRUE;
	//////////////////////////////////////////////
	//////////////////////////////////////////////
	//	E_BA_AC_OpMod01.eNightCooling
	CoolerOpMod.arrOpModVal[E_BA_AC_OpMod01.eNightCooling]				:= FALSE;
	CoolerOpMod.arrIgnoreDelayOnVal[E_BA_AC_OpMod01.eNightCooling]		:= TRUE;
	CoolerOpMod.arrIgnoreDelayOffVal[E_BA_AC_OpMod01.eNightCooling]		:= TRUE;
	CoolerOpMod.arrIgnoreFdbVal[E_BA_AC_OpMod01.eNightCooling]			:= TRUE;
	//////////////////////////////////////////////
	//////////////////////////////////////////////
	//	E_BA_AC_OpMod01.eCoolDownProtection
	CoolerOpMod.arrOpModVal[E_BA_AC_OpMod01.eCoolDownProtection]				:= FALSE;
	CoolerOpMod.arrIgnoreDelayOnVal[E_BA_AC_OpMod01.eCoolDownProtection]		:= TRUE;
	CoolerOpMod.arrIgnoreDelayOffVal[E_BA_AC_OpMod01.eCoolDownProtection]		:= TRUE;
	CoolerOpMod.arrIgnoreFdbVal[E_BA_AC_OpMod01.eCoolDownProtection]			:= TRUE;
	//////////////////////////////////////////////
	//////////////////////////////////////////////
	//	E_BA_AC_OpMod01.eOverHeatingProtection
	CoolerOpMod.arrOpModVal[E_BA_AC_OpMod01.eOverHeatingProtection]				:= TRUE;
	CoolerOpMod.arrIgnoreDelayOnVal[E_BA_AC_OpMod01.eOverHeatingProtection]		:= TRUE;
	CoolerOpMod.arrIgnoreDelayOffVal[E_BA_AC_OpMod01.eOverHeatingProtection]	:= TRUE;
	CoolerOpMod.arrIgnoreFdbVal[E_BA_AC_OpMod01.eOverHeatingProtection]			:= TRUE;
	//////////////////////////////////////////////
	//////////////////////////////////////////////
	//	E_BA_AC_OpMod01.eAlarm
	CoolerOpMod.arrOpModVal[E_BA_AC_OpMod01.eAlarm]				:= FALSE;
	CoolerOpMod.arrIgnoreDelayOnVal[E_BA_AC_OpMod01.eAlarm]		:= TRUE;
	CoolerOpMod.arrIgnoreDelayOffVal[E_BA_AC_OpMod01.eAlarm]	:= TRUE;
	CoolerOpMod.arrIgnoreFdbVal[E_BA_AC_OpMod01.eAlarm]			:= TRUE;
	//////////////////////////////////////////////
	//////////////////////////////////////////////
	//	E_BA_AC_OpMod01.eForcedVentilation
	CoolerOpMod.arrOpModVal[E_BA_AC_OpMod01.eForcedVentilation]				:= TRUE;
	CoolerOpMod.arrIgnoreDelayOnVal[E_BA_AC_OpMod01.eForcedVentilation]		:= TRUE;
	CoolerOpMod.arrIgnoreDelayOffVal[E_BA_AC_OpMod01.eForcedVentilation]	:= TRUE;
	CoolerOpMod.arrIgnoreFdbVal[E_BA_AC_OpMod01.eForcedVentilation]			:= TRUE;
	//////////////////////////////////////////////
	//////////////////////////////////////////////
	//	E_BA_AC_OpMod01.eCentralSwitchOff
	CoolerOpMod.arrOpModVal[E_BA_AC_OpMod01.eCentralSwitchOff]				:= FALSE;
	CoolerOpMod.arrIgnoreDelayOnVal[E_BA_AC_OpMod01.eCentralSwitchOff]		:= TRUE;
	CoolerOpMod.arrIgnoreDelayOffVal[E_BA_AC_OpMod01.eCentralSwitchOff]		:= TRUE;
	CoolerOpMod.arrIgnoreFdbVal[E_BA_AC_OpMod01.eCentralSwitchOff]			:= TRUE;
	//////////////////////////////////////////////
	//////////////////////////////////////////////
	//	E_BA_AC_OpMod01.eCustomer01
	CoolerOpMod.arrOpModVal[E_BA_AC_OpMod01.eCustomer01]				:= FALSE;
	CoolerOpMod.arrIgnoreDelayOnVal[E_BA_AC_OpMod01.eCustomer01]		:= TRUE;
	CoolerOpMod.arrIgnoreDelayOffVal[E_BA_AC_OpMod01.eCustomer01]		:= TRUE;
	CoolerOpMod.arrIgnoreFdbVal[E_BA_AC_OpMod01.eCustomer01]			:= TRUE;
	//////////////////////////////////////////////
	//////////////////////////////////////////////
	//	E_BA_AC_OpMod01.eCustomer02
	CoolerOpMod.arrOpModVal[E_BA_AC_OpMod01.eCustomer02]				:= FALSE;
	CoolerOpMod.arrIgnoreDelayOnVal[E_BA_AC_OpMod01.eCustomer02]		:= TRUE;
	CoolerOpMod.arrIgnoreDelayOffVal[E_BA_AC_OpMod01.eCustomer02]		:= TRUE;
	CoolerOpMod.arrIgnoreFdbVal[E_BA_AC_OpMod01.eCustomer02]			:= TRUE;
END_IF
END_METHOD

METHOD InitErc
VAR_INPUT
END_VAR
IF	ErcOpMod.bInit
THEN	
	ErcOpMod.bInit := FALSE;
	//////////////////////////////////////////////
	//////////////////////////////////////////////
	//	E_BA_AC_OpMod01.eOff;
	ErcOpMod.arrOpModVal[E_BA_AC_OpMod01.eOff]				:= FALSE;
	ErcOpMod.arrIgnoreDelayOnVal[E_BA_AC_OpMod01.eOff]		:= TRUE;
	ErcOpMod.arrIgnoreDelayOffVal[E_BA_AC_OpMod01.eOff]		:= TRUE;
	ErcOpMod.arrIgnoreFdbVal[E_BA_AC_OpMod01.eOff]			:= TRUE;	
	//////////////////////////////////////////////
	//////////////////////////////////////////////
	//	E_BA_AC_OpMod01.eOn;
	ErcOpMod.arrOpModVal[E_BA_AC_OpMod01.eOn]				:= TRUE;
	ErcOpMod.arrIgnoreDelayOnVal[E_BA_AC_OpMod01.eOn]		:= TRUE;
	ErcOpMod.arrIgnoreDelayOffVal[E_BA_AC_OpMod01.eOn]		:= TRUE;
	ErcOpMod.arrIgnoreFdbVal[E_BA_AC_OpMod01.eOn]			:= TRUE;
	//////////////////////////////////////////////
	//////////////////////////////////////////////
	//	E_BA_AC_OpMod01.eEmergency;
	ErcOpMod.arrOpModVal[E_BA_AC_OpMod01.eEmergency]				:= FALSE;
	ErcOpMod.arrIgnoreDelayOnVal[E_BA_AC_OpMod01.eEmergency]		:= TRUE;
	ErcOpMod.arrIgnoreDelayOffVal[E_BA_AC_OpMod01.eEmergency]		:= TRUE;
	ErcOpMod.arrIgnoreFdbVal[E_BA_AC_OpMod01.eEmergency]			:= TRUE;
	//////////////////////////////////////////////
	//////////////////////////////////////////////
	//	E_BA_AC_OpMod01.eFrost;
	ErcOpMod.arrOpModVal[E_BA_AC_OpMod01.eFrost]				:= FALSE;
	ErcOpMod.arrIgnoreDelayOnVal[E_BA_AC_OpMod01.eFrost]		:= TRUE;
	ErcOpMod.arrIgnoreDelayOffVal[E_BA_AC_OpMod01.eFrost]		:= TRUE;
	ErcOpMod.arrIgnoreFdbVal[E_BA_AC_OpMod01.eFrost]			:= TRUE;
	//////////////////////////////////////////////
	//////////////////////////////////////////////
	//	E_BA_AC_OpMod01.eSmokeExtractionProgramm;
	ErcOpMod.arrOpModVal[E_BA_AC_OpMod01.eSmokeExtractionProgram]				:= FALSE;
	ErcOpMod.arrIgnoreDelayOnVal[E_BA_AC_OpMod01.eSmokeExtractionProgram]		:= TRUE;
	ErcOpMod.arrIgnoreDelayOffVal[E_BA_AC_OpMod01.eSmokeExtractionProgram]		:= TRUE;
	ErcOpMod.arrIgnoreFdbVal[E_BA_AC_OpMod01.eSmokeExtractionProgram]			:= TRUE;
	//////////////////////////////////////////////
	//////////////////////////////////////////////
	//	E_BA_AC_OpMod01.eSmokeExtractionSupplyAir;
	ErcOpMod.arrOpModVal[E_BA_AC_OpMod01.eSmokeExtractionSupplyAir]				:= FALSE;
	ErcOpMod.arrIgnoreDelayOnVal[E_BA_AC_OpMod01.eSmokeExtractionSupplyAir]		:= TRUE;
	ErcOpMod.arrIgnoreDelayOffVal[E_BA_AC_OpMod01.eSmokeExtractionSupplyAir]	:= TRUE;
	ErcOpMod.arrIgnoreFdbVal[E_BA_AC_OpMod01.eSmokeExtractionSupplyAir]			:= TRUE;
	//////////////////////////////////////////////
	//////////////////////////////////////////////
	//	E_BA_AC_OpMod01.eSmokeExtractionExhaustAir;
	ErcOpMod.arrOpModVal[E_BA_AC_OpMod01.eSmokeExtractionExhaustAir]				:= FALSE;
	ErcOpMod.arrIgnoreDelayOnVal[E_BA_AC_OpMod01.eSmokeExtractionExhaustAir]		:= TRUE;
	ErcOpMod.arrIgnoreDelayOffVal[E_BA_AC_OpMod01.eSmokeExtractionExhaustAir]		:= TRUE;
	ErcOpMod.arrIgnoreFdbVal[E_BA_AC_OpMod01.eSmokeExtractionExhaustAir]			:= TRUE;
	//////////////////////////////////////////////
	//////////////////////////////////////////////
	//	E_BA_AC_OpMod01.eFire;
	ErcOpMod.arrOpModVal[E_BA_AC_OpMod01.eFire]				:= FALSE;
	ErcOpMod.arrIgnoreDelayOnVal[E_BA_AC_OpMod01.eFire]		:= TRUE;
	ErcOpMod.arrIgnoreDelayOffVal[E_BA_AC_OpMod01.eFire]	:= TRUE;
	ErcOpMod.arrIgnoreFdbVal[E_BA_AC_OpMod01.eFire]			:= TRUE;
	//////////////////////////////////////////////
	//////////////////////////////////////////////
	//	E_BA_AC_OpMod01.eNightCooling;
	ErcOpMod.arrOpModVal[E_BA_AC_OpMod01.eNightCooling]				:= FALSE;
	ErcOpMod.arrIgnoreDelayOnVal[E_BA_AC_OpMod01.eNightCooling]		:= TRUE;
	ErcOpMod.arrIgnoreDelayOffVal[E_BA_AC_OpMod01.eNightCooling]	:= TRUE;
	ErcOpMod.arrIgnoreFdbVal[E_BA_AC_OpMod01.eNightCooling]			:= TRUE;
	//////////////////////////////////////////////
	//////////////////////////////////////////////
	//	E_BA_AC_OpMod01.eCoolDownProtection;
	ErcOpMod.arrOpModVal[E_BA_AC_OpMod01.eCoolDownProtection]				:= TRUE;
	ErcOpMod.arrIgnoreDelayOnVal[E_BA_AC_OpMod01.eCoolDownProtection]		:= TRUE;
	ErcOpMod.arrIgnoreDelayOffVal[E_BA_AC_OpMod01.eCoolDownProtection]		:= TRUE;
	ErcOpMod.arrIgnoreFdbVal[E_BA_AC_OpMod01.eCoolDownProtection]			:= TRUE;
	//////////////////////////////////////////////
	//////////////////////////////////////////////
	//	E_BA_AC_OpMod01.eOverHeatingProtection;
	ErcOpMod.arrOpModVal[E_BA_AC_OpMod01.eOverHeatingProtection]			:= TRUE;
	ErcOpMod.arrIgnoreDelayOnVal[E_BA_AC_OpMod01.eOverHeatingProtection]	:= TRUE;
	ErcOpMod.arrIgnoreDelayOffVal[E_BA_AC_OpMod01.eOverHeatingProtection]	:= TRUE;
	ErcOpMod.arrIgnoreFdbVal[E_BA_AC_OpMod01.eOverHeatingProtection]		:= TRUE;
	//////////////////////////////////////////////
	//////////////////////////////////////////////
	//	E_BA_AC_OpMod01.eAlarm;
	ErcOpMod.arrOpModVal[E_BA_AC_OpMod01.eAlarm]				:= FALSE;
	ErcOpMod.arrIgnoreDelayOnVal[E_BA_AC_OpMod01.eAlarm]		:= TRUE;
	ErcOpMod.arrIgnoreDelayOffVal[E_BA_AC_OpMod01.eAlarm]		:= TRUE;
	ErcOpMod.arrIgnoreFdbVal[E_BA_AC_OpMod01.eAlarm]			:= TRUE;
	//////////////////////////////////////////////
	//////////////////////////////////////////////
	//	E_BA_AC_OpMod01.eForcedVentilation;
	ErcOpMod.arrOpModVal[E_BA_AC_OpMod01.eForcedVentilation]				:= TRUE;
	ErcOpMod.arrIgnoreDelayOnVal[E_BA_AC_OpMod01.eForcedVentilation]		:= TRUE;
	ErcOpMod.arrIgnoreDelayOffVal[E_BA_AC_OpMod01.eForcedVentilation]		:= TRUE;
	ErcOpMod.arrIgnoreFdbVal[E_BA_AC_OpMod01.eForcedVentilation]			:= TRUE;
	//////////////////////////////////////////////
	//////////////////////////////////////////////
	//	E_BA_AC_OpMod01.eCentralSwitchOff;
	ErcOpMod.arrOpModVal[E_BA_AC_OpMod01.eCentralSwitchOff]				:= FALSE;
	ErcOpMod.arrIgnoreDelayOnVal[E_BA_AC_OpMod01.eCentralSwitchOff]		:= TRUE;
	ErcOpMod.arrIgnoreDelayOffVal[E_BA_AC_OpMod01.eCentralSwitchOff]	:= TRUE;
	ErcOpMod.arrIgnoreFdbVal[E_BA_AC_OpMod01.eCentralSwitchOff]			:= TRUE;
	//////////////////////////////////////////////
	//////////////////////////////////////////////
	//	E_BA_AC_OpMod01.eCustomer01;
	ErcOpMod.arrOpModVal[E_BA_AC_OpMod01.eCustomer01]				:= FALSE;
	ErcOpMod.arrIgnoreDelayOnVal[E_BA_AC_OpMod01.eCustomer01]		:= TRUE;
	ErcOpMod.arrIgnoreDelayOffVal[E_BA_AC_OpMod01.eCustomer01]		:= TRUE;
	ErcOpMod.arrIgnoreFdbVal[E_BA_AC_OpMod01.eCustomer01]			:= TRUE;
	//////////////////////////////////////////////
	//////////////////////////////////////////////
	//	E_BA_AC_OpMod01.eCustomer02;
	ErcOpMod.arrOpModVal[E_BA_AC_OpMod01.eCustomer02]				:= FALSE;
	ErcOpMod.arrIgnoreDelayOnVal[E_BA_AC_OpMod01.eCustomer02]		:= TRUE;
	ErcOpMod.arrIgnoreDelayOffVal[E_BA_AC_OpMod01.eCustomer02]		:= TRUE;
	ErcOpMod.arrIgnoreFdbVal[E_BA_AC_OpMod01.eCustomer02]			:= TRUE;
END_IF
END_METHOD

METHOD InitExhADmp
VAR_INPUT
END_VAR
IF	ExhADmpOpMod.bInit
THEN	
	ExhADmpOpMod.bInit := FALSE;
	//////////////////////////////////////////////
	//////////////////////////////////////////////
	//	E_BA_AC_OpMod01.eOff
	ExhADmpOpMod.arrOpModVal[E_BA_AC_OpMod01.eOff]				:= FALSE;
	ExhADmpOpMod.arrIgnoreDelayOnVal[E_BA_AC_OpMod01.eOff]		:= TRUE;
	ExhADmpOpMod.arrIgnoreDelayOffVal[E_BA_AC_OpMod01.eOff]		:= FALSE;
	ExhADmpOpMod.arrIgnoreFdbVal[E_BA_AC_OpMod01.eOff]			:= TRUE;
	//////////////////////////////////////////////
	//////////////////////////////////////////////
	//	E_BA_AC_OpMod01.eOn;
	ExhADmpOpMod.arrOpModVal[E_BA_AC_OpMod01.eOn]				:= TRUE;
	ExhADmpOpMod.arrIgnoreDelayOnVal[E_BA_AC_OpMod01.eOn]		:= TRUE;
	ExhADmpOpMod.arrIgnoreDelayOffVal[E_BA_AC_OpMod01.eOn]		:= TRUE;
	ExhADmpOpMod.arrIgnoreFdbVal[E_BA_AC_OpMod01.eOn]			:= FALSE;
	//////////////////////////////////////////////
	//////////////////////////////////////////////
	//	E_BA_AC_OpMod01.eEmergency;
	ExhADmpOpMod.arrOpModVal[E_BA_AC_OpMod01.eEmergency]				:= FALSE;
	ExhADmpOpMod.arrIgnoreDelayOnVal[E_BA_AC_OpMod01.eEmergency]		:= TRUE;
	ExhADmpOpMod.arrIgnoreDelayOffVal[E_BA_AC_OpMod01.eEmergency]		:= TRUE;
	ExhADmpOpMod.arrIgnoreFdbVal[E_BA_AC_OpMod01.eEmergency]			:= TRUE;
	//////////////////////////////////////////////
	//////////////////////////////////////////////
	//	E_BA_AC_OpMod01.eFrost;
	ExhADmpOpMod.arrOpModVal[E_BA_AC_OpMod01.eFrost]				:= FALSE;
	ExhADmpOpMod.arrIgnoreDelayOnVal[E_BA_AC_OpMod01.eFrost]		:= TRUE;
	ExhADmpOpMod.arrIgnoreDelayOffVal[E_BA_AC_OpMod01.eFrost]		:= FALSE;
	ExhADmpOpMod.arrIgnoreFdbVal[E_BA_AC_OpMod01.eFrost]			:= TRUE;
	//////////////////////////////////////////////
	//////////////////////////////////////////////
	//	E_BA_AC_OpMod01.eSmokeExtractionProgramm;
	ExhADmpOpMod.arrOpModVal[E_BA_AC_OpMod01.eSmokeExtractionProgram]				:= TRUE;
	ExhADmpOpMod.arrIgnoreDelayOnVal[E_BA_AC_OpMod01.eSmokeExtractionProgram]		:= TRUE;
	ExhADmpOpMod.arrIgnoreDelayOffVal[E_BA_AC_OpMod01.eSmokeExtractionProgram]		:= TRUE;
	ExhADmpOpMod.arrIgnoreFdbVal[E_BA_AC_OpMod01.eSmokeExtractionProgram]			:= TRUE;
	//////////////////////////////////////////////
	//////////////////////////////////////////////
	//	E_BA_AC_OpMod01.eSmokeExtractionSupplyAir;
	ExhADmpOpMod.arrOpModVal[E_BA_AC_OpMod01.eSmokeExtractionSupplyAir]				:= FALSE;
	ExhADmpOpMod.arrIgnoreDelayOnVal[E_BA_AC_OpMod01.eSmokeExtractionSupplyAir]		:= TRUE;
	ExhADmpOpMod.arrIgnoreDelayOffVal[E_BA_AC_OpMod01.eSmokeExtractionSupplyAir]	:= FALSE;
	ExhADmpOpMod.arrIgnoreFdbVal[E_BA_AC_OpMod01.eSmokeExtractionSupplyAir]			:= TRUE;
	//////////////////////////////////////////////
	//////////////////////////////////////////////
	//	E_BA_AC_OpMod01.eSmokeExtractionExhaustAir;
	ExhADmpOpMod.arrOpModVal[E_BA_AC_OpMod01.eSmokeExtractionExhaustAir]				:= TRUE;
	ExhADmpOpMod.arrIgnoreDelayOnVal[E_BA_AC_OpMod01.eSmokeExtractionExhaustAir]		:= TRUE;
	ExhADmpOpMod.arrIgnoreDelayOffVal[E_BA_AC_OpMod01.eSmokeExtractionExhaustAir]		:= TRUE;
	ExhADmpOpMod.arrIgnoreFdbVal[E_BA_AC_OpMod01.eSmokeExtractionExhaustAir]			:= TRUE;
	//////////////////////////////////////////////
	//////////////////////////////////////////////
	//	E_BA_AC_OpMod01.eFire;
	ExhADmpOpMod.arrOpModVal[E_BA_AC_OpMod01.eFire]				:= FALSE;
	ExhADmpOpMod.arrIgnoreDelayOnVal[E_BA_AC_OpMod01.eFire]		:= TRUE;
	ExhADmpOpMod.arrIgnoreDelayOffVal[E_BA_AC_OpMod01.eFire]	:= TRUE;
	ExhADmpOpMod.arrIgnoreFdbVal[E_BA_AC_OpMod01.eFire]			:= TRUE;
	//////////////////////////////////////////////
	//////////////////////////////////////////////
	//	E_BA_AC_OpMod01.eNightCooling;
	ExhADmpOpMod.arrOpModVal[E_BA_AC_OpMod01.eNightCooling]				:= TRUE;
	ExhADmpOpMod.arrIgnoreDelayOnVal[E_BA_AC_OpMod01.eNightCooling]		:= TRUE;
	ExhADmpOpMod.arrIgnoreDelayOffVal[E_BA_AC_OpMod01.eNightCooling]	:= TRUE;
	ExhADmpOpMod.arrIgnoreFdbVal[E_BA_AC_OpMod01.eNightCooling]			:= FALSE;
	//////////////////////////////////////////////
	//////////////////////////////////////////////
	//	E_BA_AC_OpMod01.eCoolDownProtection;
	ExhADmpOpMod.arrOpModVal[E_BA_AC_OpMod01.eCoolDownProtection]				:= TRUE;
	ExhADmpOpMod.arrIgnoreDelayOnVal[E_BA_AC_OpMod01.eCoolDownProtection]		:= TRUE;
	ExhADmpOpMod.arrIgnoreDelayOffVal[E_BA_AC_OpMod01.eCoolDownProtection]		:= TRUE;
	ExhADmpOpMod.arrIgnoreFdbVal[E_BA_AC_OpMod01.eCoolDownProtection]			:= FALSE;
	//////////////////////////////////////////////
	//////////////////////////////////////////////
	//	E_BA_AC_OpMod01.eOverHeatingProtection;
	ExhADmpOpMod.arrOpModVal[E_BA_AC_OpMod01.eOverHeatingProtection]				:= TRUE;
	ExhADmpOpMod.arrIgnoreDelayOnVal[E_BA_AC_OpMod01.eOverHeatingProtection]		:= TRUE;
	ExhADmpOpMod.arrIgnoreDelayOffVal[E_BA_AC_OpMod01.eOverHeatingProtection]		:= TRUE;
	ExhADmpOpMod.arrIgnoreFdbVal[E_BA_AC_OpMod01.eOverHeatingProtection]			:= FALSE;
	//////////////////////////////////////////////
	//////////////////////////////////////////////
	//	E_BA_AC_OpMod01.eAlarm;
	ExhADmpOpMod.arrOpModVal[E_BA_AC_OpMod01.eAlarm]				:= FALSE;
	ExhADmpOpMod.arrIgnoreDelayOnVal[E_BA_AC_OpMod01.eAlarm]		:= TRUE;
	ExhADmpOpMod.arrIgnoreDelayOffVal[E_BA_AC_OpMod01.eAlarm]		:= FALSE;
	ExhADmpOpMod.arrIgnoreFdbVal[E_BA_AC_OpMod01.eAlarm]			:= TRUE;
	//////////////////////////////////////////////
	//////////////////////////////////////////////
	//	E_BA_AC_OpMod01.eForcedVentilation;
	ExhADmpOpMod.arrOpModVal[E_BA_AC_OpMod01.eForcedVentilation]				:= TRUE;
	ExhADmpOpMod.arrIgnoreDelayOnVal[E_BA_AC_OpMod01.eForcedVentilation]		:= TRUE;
	ExhADmpOpMod.arrIgnoreDelayOffVal[E_BA_AC_OpMod01.eForcedVentilation]		:= TRUE;
	ExhADmpOpMod.arrIgnoreFdbVal[E_BA_AC_OpMod01.eForcedVentilation]			:= FALSE;
	//////////////////////////////////////////////
	//////////////////////////////////////////////
	//	E_BA_AC_OpMod01.eCentralSwitchOff;
	ExhADmpOpMod.arrOpModVal[E_BA_AC_OpMod01.eCentralSwitchOff]				:= FALSE;
	ExhADmpOpMod.arrIgnoreDelayOnVal[E_BA_AC_OpMod01.eCentralSwitchOff]		:= TRUE;
	ExhADmpOpMod.arrIgnoreDelayOffVal[E_BA_AC_OpMod01.eCentralSwitchOff]	:= FALSE;
	ExhADmpOpMod.arrIgnoreFdbVal[E_BA_AC_OpMod01.eCentralSwitchOff]			:= TRUE;
	//////////////////////////////////////////////
	//////////////////////////////////////////////
	//	E_BA_AC_OpMod01.eCustomer01;
	ExhADmpOpMod.arrOpModVal[E_BA_AC_OpMod01.eCustomer01]				:= FALSE;
	ExhADmpOpMod.arrIgnoreDelayOnVal[E_BA_AC_OpMod01.eCustomer01]		:= TRUE;
	ExhADmpOpMod.arrIgnoreDelayOffVal[E_BA_AC_OpMod01.eCustomer01]		:= FALSE;
	ExhADmpOpMod.arrIgnoreFdbVal[E_BA_AC_OpMod01.eCustomer01]			:= TRUE;
	//////////////////////////////////////////////
	//////////////////////////////////////////////
	//	E_BA_AC_OpMod01.eCustomer02;
	ExhADmpOpMod.arrOpModVal[E_BA_AC_OpMod01.eCustomer02]				:= FALSE;
	ExhADmpOpMod.arrIgnoreDelayOnVal[E_BA_AC_OpMod01.eCustomer02]		:= TRUE;
	ExhADmpOpMod.arrIgnoreDelayOffVal[E_BA_AC_OpMod01.eCustomer02]		:= FALSE;
	ExhADmpOpMod.arrIgnoreFdbVal[E_BA_AC_OpMod01.eCustomer02]			:= TRUE;
END_IF
END_METHOD

METHOD InitExtAFan
VAR_INPUT
END_VAR
IF	ExtAFanOpMod.bInit
THEN	
	ExtAFanOpMod.bInit := FALSE;
	//////////////////////////////////////////////
	//////////////////////////////////////////////
	//	E_BA_AC_OpMod01.eOff;
	ExtAFanOpMod.arrOpModVal[E_BA_AC_OpMod01.eOff]				:= E_BA_Mdlt.eOff;
	ExtAFanOpMod.arrIgnoreDelayOnVal[E_BA_AC_OpMod01.eOff]		:= TRUE;
	ExtAFanOpMod.arrIgnoreDelayOffVal[E_BA_AC_OpMod01.eOff]		:= TRUE;
	ExtAFanOpMod.arrIgnoreFdbVal[E_BA_AC_OpMod01.eOff]			:= TRUE;
	//////////////////////////////////////////////
	//////////////////////////////////////////////
	//	E_BA_AC_OpMod01.eOn;
	ExtAFanOpMod.arrOpModVal[E_BA_AC_OpMod01.eOn]				:= E_BA_Mdlt.eOn;
	ExtAFanOpMod.arrIgnoreDelayOnVal[E_BA_AC_OpMod01.eOn]		:= TRUE;
	ExtAFanOpMod.arrIgnoreDelayOffVal[E_BA_AC_OpMod01.eOn]		:= TRUE;
	ExtAFanOpMod.arrIgnoreFdbVal[E_BA_AC_OpMod01.eOn]			:= TRUE;
	//////////////////////////////////////////////
	//////////////////////////////////////////////
	//	E_BA_AC_OpMod01.eEmergency;
	ExtAFanOpMod.arrOpModVal[E_BA_AC_OpMod01.eEmergency]				:= E_BA_Mdlt.eOff;
	ExtAFanOpMod.arrIgnoreDelayOnVal[E_BA_AC_OpMod01.eEmergency]		:= TRUE;
	ExtAFanOpMod.arrIgnoreDelayOffVal[E_BA_AC_OpMod01.eEmergency]		:= TRUE;
	ExtAFanOpMod.arrIgnoreFdbVal[E_BA_AC_OpMod01.eEmergency]			:= TRUE;
	//////////////////////////////////////////////
	//////////////////////////////////////////////
	//	E_BA_AC_OpMod01.eFrost;
	ExtAFanOpMod.arrOpModVal[E_BA_AC_OpMod01.eFrost]				:= E_BA_Mdlt.eOff;
	ExtAFanOpMod.arrIgnoreDelayOnVal[E_BA_AC_OpMod01.eFrost]		:= TRUE;
	ExtAFanOpMod.arrIgnoreDelayOffVal[E_BA_AC_OpMod01.eFrost]		:= TRUE;
	ExtAFanOpMod.arrIgnoreFdbVal[E_BA_AC_OpMod01.eFrost]			:= TRUE;
	//////////////////////////////////////////////
	//////////////////////////////////////////////
	//	E_BA_AC_OpMod01.eSmokeExtractionProgramm;
	ExtAFanOpMod.arrOpModVal[E_BA_AC_OpMod01.eSmokeExtractionProgram]				:= E_BA_Mdlt.eOn;
	ExtAFanOpMod.arrIgnoreDelayOnVal[E_BA_AC_OpMod01.eSmokeExtractionProgram]		:= TRUE;
	ExtAFanOpMod.arrIgnoreDelayOffVal[E_BA_AC_OpMod01.eSmokeExtractionProgram]		:= TRUE;
	ExtAFanOpMod.arrIgnoreFdbVal[E_BA_AC_OpMod01.eSmokeExtractionProgram]			:= TRUE;
	//////////////////////////////////////////////
	//////////////////////////////////////////////
	//	E_BA_AC_OpMod01.eSmokeExtractionSupplyAir;
	ExtAFanOpMod.arrOpModVal[E_BA_AC_OpMod01.eSmokeExtractionSupplyAir]				:= E_BA_Mdlt.eOff;
	ExtAFanOpMod.arrIgnoreDelayOnVal[E_BA_AC_OpMod01.eSmokeExtractionSupplyAir]		:= TRUE;
	ExtAFanOpMod.arrIgnoreDelayOffVal[E_BA_AC_OpMod01.eSmokeExtractionSupplyAir]	:= TRUE;
	ExtAFanOpMod.arrIgnoreFdbVal[E_BA_AC_OpMod01.eSmokeExtractionSupplyAir]			:= TRUE;
	//////////////////////////////////////////////
	//////////////////////////////////////////////
	//	E_BA_AC_OpMod01.eSmokeExtractionExhaustAir;
	ExtAFanOpMod.arrOpModVal[E_BA_AC_OpMod01.eSmokeExtractionExhaustAir]				:= E_BA_Mdlt.eOn;
	ExtAFanOpMod.arrIgnoreDelayOnVal[E_BA_AC_OpMod01.eSmokeExtractionExhaustAir]		:= TRUE;
	ExtAFanOpMod.arrIgnoreDelayOffVal[E_BA_AC_OpMod01.eSmokeExtractionExhaustAir]		:= TRUE;
	ExtAFanOpMod.arrIgnoreFdbVal[E_BA_AC_OpMod01.eSmokeExtractionExhaustAir]			:= TRUE;
	//////////////////////////////////////////////
	//////////////////////////////////////////////
	//	E_BA_AC_OpMod01.eFire;
	ExtAFanOpMod.arrOpModVal[E_BA_AC_OpMod01.eFire]				:= E_BA_Mdlt.eOff;
	ExtAFanOpMod.arrIgnoreDelayOnVal[E_BA_AC_OpMod01.eFire]		:= TRUE;
	ExtAFanOpMod.arrIgnoreDelayOffVal[E_BA_AC_OpMod01.eFire]	:= TRUE;
	ExtAFanOpMod.arrIgnoreFdbVal[E_BA_AC_OpMod01.eFire]			:= TRUE;
	//////////////////////////////////////////////
	//////////////////////////////////////////////
	//	E_BA_AC_OpMod01.eNightCooling;
	ExtAFanOpMod.arrOpModVal[E_BA_AC_OpMod01.eNightCooling]				:= E_BA_Mdlt.eOn;
	ExtAFanOpMod.arrIgnoreDelayOnVal[E_BA_AC_OpMod01.eNightCooling]		:= TRUE;
	ExtAFanOpMod.arrIgnoreDelayOffVal[E_BA_AC_OpMod01.eNightCooling]	:= TRUE;
	ExtAFanOpMod.arrIgnoreFdbVal[E_BA_AC_OpMod01.eNightCooling]			:= TRUE;
	//////////////////////////////////////////////
	//////////////////////////////////////////////
	//	E_BA_AC_OpMod01.eCoolDownProtection;
	ExtAFanOpMod.arrOpModVal[E_BA_AC_OpMod01.eCoolDownProtection]				:= E_BA_Mdlt.eOn;
	ExtAFanOpMod.arrIgnoreDelayOnVal[E_BA_AC_OpMod01.eCoolDownProtection]		:= TRUE;
	ExtAFanOpMod.arrIgnoreDelayOffVal[E_BA_AC_OpMod01.eCoolDownProtection]		:= TRUE;
	ExtAFanOpMod.arrIgnoreFdbVal[E_BA_AC_OpMod01.eCoolDownProtection]			:= TRUE;
	//////////////////////////////////////////////
	//////////////////////////////////////////////
	//	E_BA_AC_OpMod01.eOverHeatingProtection;
	ExtAFanOpMod.arrOpModVal[E_BA_AC_OpMod01.eOverHeatingProtection]				:= E_BA_Mdlt.eOn;
	ExtAFanOpMod.arrIgnoreDelayOnVal[E_BA_AC_OpMod01.eOverHeatingProtection]		:= TRUE;
	ExtAFanOpMod.arrIgnoreDelayOffVal[E_BA_AC_OpMod01.eOverHeatingProtection]		:= TRUE;
	ExtAFanOpMod.arrIgnoreFdbVal[E_BA_AC_OpMod01.eOverHeatingProtection]			:= TRUE;
	//////////////////////////////////////////////
	//////////////////////////////////////////////
	//	E_BA_AC_OpMod01.eAlarm;
	ExtAFanOpMod.arrOpModVal[E_BA_AC_OpMod01.eAlarm]				:= E_BA_Mdlt.eOff;
	ExtAFanOpMod.arrIgnoreDelayOnVal[E_BA_AC_OpMod01.eAlarm]		:= TRUE;
	ExtAFanOpMod.arrIgnoreDelayOffVal[E_BA_AC_OpMod01.eAlarm]		:= TRUE;
	ExtAFanOpMod.arrIgnoreFdbVal[E_BA_AC_OpMod01.eAlarm]			:= TRUE;
	//////////////////////////////////////////////
	//////////////////////////////////////////////
	//	E_BA_AC_OpMod01.eForcedVentilation;
	ExtAFanOpMod.arrOpModVal[E_BA_AC_OpMod01.eForcedVentilation]				:= E_BA_Mdlt.eOn;
	ExtAFanOpMod.arrIgnoreDelayOnVal[E_BA_AC_OpMod01.eForcedVentilation]		:= TRUE;
	ExtAFanOpMod.arrIgnoreDelayOffVal[E_BA_AC_OpMod01.eForcedVentilation]		:= TRUE;
	ExtAFanOpMod.arrIgnoreFdbVal[E_BA_AC_OpMod01.eForcedVentilation]			:= TRUE;
	//////////////////////////////////////////////
	//////////////////////////////////////////////
	//	E_BA_AC_OpMod01.eCentralSwitchOff;
	ExtAFanOpMod.arrOpModVal[E_BA_AC_OpMod01.eCentralSwitchOff]				:= E_BA_Mdlt.eOff;
	ExtAFanOpMod.arrIgnoreDelayOnVal[E_BA_AC_OpMod01.eCentralSwitchOff]		:= TRUE;
	ExtAFanOpMod.arrIgnoreDelayOffVal[E_BA_AC_OpMod01.eCentralSwitchOff]	:= TRUE;
	ExtAFanOpMod.arrIgnoreFdbVal[E_BA_AC_OpMod01.eCentralSwitchOff]			:= TRUE;
	//////////////////////////////////////////////
	//////////////////////////////////////////////
	//	E_BA_AC_OpMod01.eCustomer01;
	ExtAFanOpMod.arrOpModVal[E_BA_AC_OpMod01.eCustomer01]				:= E_BA_Mdlt.eOff;
	ExtAFanOpMod.arrIgnoreDelayOnVal[E_BA_AC_OpMod01.eCustomer01]		:= TRUE;
	ExtAFanOpMod.arrIgnoreDelayOffVal[E_BA_AC_OpMod01.eCustomer01]		:= TRUE;
	ExtAFanOpMod.arrIgnoreFdbVal[E_BA_AC_OpMod01.eCustomer01]			:= TRUE;
	//////////////////////////////////////////////
	//////////////////////////////////////////////
	//	E_BA_AC_OpMod01.eCustomer02;
	ExtAFanOpMod.arrOpModVal[E_BA_AC_OpMod01.eCustomer02]				:= E_BA_Mdlt.eOff;
	ExtAFanOpMod.arrIgnoreDelayOnVal[E_BA_AC_OpMod01.eCustomer02]		:= TRUE;
	ExtAFanOpMod.arrIgnoreDelayOffVal[E_BA_AC_OpMod01.eCustomer02]		:= TRUE;
	ExtAFanOpMod.arrIgnoreFdbVal[E_BA_AC_OpMod01.eCustomer02]			:= TRUE;
END_IF
END_METHOD

METHOD InitOuADmp
VAR_INPUT
END_VAR
IF	OuADmpOpMod.bInit
THEN	
	OuADmpOpMod.bInit := FALSE;
	//////////////////////////////////////////////
	//////////////////////////////////////////////
	//	E_BA_AC_OpMod01.eOff;
	OuADmpOpMod.arrOpModVal[E_BA_AC_OpMod01.eOff]				:= FALSE;
	OuADmpOpMod.arrIgnoreDelayOnVal[E_BA_AC_OpMod01.eOff]		:= TRUE;
	OuADmpOpMod.arrIgnoreDelayOffVal[E_BA_AC_OpMod01.eOff]		:= FALSE;
	OuADmpOpMod.arrIgnoreFdbVal[E_BA_AC_OpMod01.eOff]			:= TRUE;
	//////////////////////////////////////////////
	//////////////////////////////////////////////
	//	E_BA_AC_OpMod01.eOn;
	OuADmpOpMod.arrOpModVal[E_BA_AC_OpMod01.eOn]				:= TRUE;
	OuADmpOpMod.arrIgnoreDelayOnVal[E_BA_AC_OpMod01.eOn]		:= TRUE;
	OuADmpOpMod.arrIgnoreDelayOffVal[E_BA_AC_OpMod01.eOn]	:= TRUE;
	OuADmpOpMod.arrIgnoreFdbVal[E_BA_AC_OpMod01.eOn]			:= FALSE;
	//////////////////////////////////////////////
	//////////////////////////////////////////////	
	//	E_BA_AC_OpMod01.eEmergency;
	OuADmpOpMod.arrOpModVal[E_BA_AC_OpMod01.eEmergency]				:= FALSE;
	OuADmpOpMod.arrIgnoreDelayOnVal[E_BA_AC_OpMod01.eEmergency]		:= TRUE;
	OuADmpOpMod.arrIgnoreDelayOffVal[E_BA_AC_OpMod01.eEmergency]		:= FALSE;
	OuADmpOpMod.arrIgnoreFdbVal[E_BA_AC_OpMod01.eEmergency]			:= TRUE;
	//////////////////////////////////////////////
	//////////////////////////////////////////////
	//	E_BA_AC_OpMod01.eFrost;
	OuADmpOpMod.arrOpModVal[E_BA_AC_OpMod01.eFrost]				:= FALSE;
	OuADmpOpMod.arrIgnoreDelayOnVal[E_BA_AC_OpMod01.eFrost]		:= TRUE;
	OuADmpOpMod.arrIgnoreDelayOffVal[E_BA_AC_OpMod01.eFrost]		:= FALSE;
	OuADmpOpMod.arrIgnoreFdbVal[E_BA_AC_OpMod01.eFrost]			:= TRUE;
	//////////////////////////////////////////////
	//////////////////////////////////////////////
	//	E_BA_AC_OpMod01.eSmokeExtractionProgram;
	OuADmpOpMod.arrOpModVal[E_BA_AC_OpMod01.eSmokeExtractionProgram]				:= TRUE;
	OuADmpOpMod.arrIgnoreDelayOnVal[E_BA_AC_OpMod01.eSmokeExtractionProgram]		:= TRUE;
	OuADmpOpMod.arrIgnoreDelayOffVal[E_BA_AC_OpMod01.eSmokeExtractionProgram]		:= TRUE;
	OuADmpOpMod.arrIgnoreFdbVal[E_BA_AC_OpMod01.eSmokeExtractionProgram]			:= FALSE;
	//////////////////////////////////////////////
	//////////////////////////////////////////////
	//	E_BA_AC_OpMod01.eSmokeExtractionSupplyAir;
	OuADmpOpMod.arrOpModVal[E_BA_AC_OpMod01.eSmokeExtractionSupplyAir]				:= TRUE;
	OuADmpOpMod.arrIgnoreDelayOnVal[E_BA_AC_OpMod01.eSmokeExtractionSupplyAir]		:= TRUE;
	OuADmpOpMod.arrIgnoreDelayOffVal[E_BA_AC_OpMod01.eSmokeExtractionSupplyAir]		:= TRUE;
	OuADmpOpMod.arrIgnoreFdbVal[E_BA_AC_OpMod01.eSmokeExtractionSupplyAir]			:= FALSE;
	//////////////////////////////////////////////
	//////////////////////////////////////////////	
	//	E_BA_AC_OpMod01.eSmokeExtractionExhaustAir;
	OuADmpOpMod.arrOpModVal[E_BA_AC_OpMod01.eSmokeExtractionExhaustAir]				:= FALSE;
	OuADmpOpMod.arrIgnoreDelayOnVal[E_BA_AC_OpMod01.eSmokeExtractionExhaustAir]		:= TRUE;
	OuADmpOpMod.arrIgnoreDelayOffVal[E_BA_AC_OpMod01.eSmokeExtractionExhaustAir]		:= FALSE;
	OuADmpOpMod.arrIgnoreFdbVal[E_BA_AC_OpMod01.eSmokeExtractionExhaustAir]			:= TRUE;
	//////////////////////////////////////////////
	//////////////////////////////////////////////
	//	E_BA_AC_OpMod01.eFire;
	OuADmpOpMod.arrOpModVal[E_BA_AC_OpMod01.eFire]				:= FALSE;
	OuADmpOpMod.arrIgnoreDelayOnVal[E_BA_AC_OpMod01.eFire]		:= TRUE;
	OuADmpOpMod.arrIgnoreDelayOffVal[E_BA_AC_OpMod01.eFire]		:= TRUE;
	OuADmpOpMod.arrIgnoreFdbVal[E_BA_AC_OpMod01.eFire]			:= TRUE;
	//////////////////////////////////////////////
	//////////////////////////////////////////////
	//	E_BA_AC_OpMod01.eNightCooling;
	OuADmpOpMod.arrOpModVal[E_BA_AC_OpMod01.eNightCooling]				:= TRUE;
	OuADmpOpMod.arrIgnoreDelayOnVal[E_BA_AC_OpMod01.eNightCooling]		:= TRUE;
	OuADmpOpMod.arrIgnoreDelayOffVal[E_BA_AC_OpMod01.eNightCooling]		:= TRUE;
	OuADmpOpMod.arrIgnoreFdbVal[E_BA_AC_OpMod01.eNightCooling]			:= FALSE;
	//////////////////////////////////////////////
	//////////////////////////////////////////////
	//	E_BA_AC_OpMod01.eCoolDownProtection;
	OuADmpOpMod.arrOpModVal[E_BA_AC_OpMod01.eCoolDownProtection]				:= TRUE;
	OuADmpOpMod.arrIgnoreDelayOnVal[E_BA_AC_OpMod01.eCoolDownProtection]		:= TRUE;
	OuADmpOpMod.arrIgnoreDelayOffVal[E_BA_AC_OpMod01.eCoolDownProtection]	:= TRUE;
	OuADmpOpMod.arrIgnoreFdbVal[E_BA_AC_OpMod01.eCoolDownProtection]			:= FALSE;
	//////////////////////////////////////////////
	//////////////////////////////////////////////
	//	E_BA_AC_OpMod01.eOverHeatingProtection;
	OuADmpOpMod.arrOpModVal[E_BA_AC_OpMod01.eOverHeatingProtection]				:= TRUE;
	OuADmpOpMod.arrIgnoreDelayOnVal[E_BA_AC_OpMod01.eOverHeatingProtection]		:= TRUE;
	OuADmpOpMod.arrIgnoreDelayOffVal[E_BA_AC_OpMod01.eOverHeatingProtection]		:= TRUE;
	OuADmpOpMod.arrIgnoreFdbVal[E_BA_AC_OpMod01.eOverHeatingProtection]			:= FALSE;
	//////////////////////////////////////////////
	//////////////////////////////////////////////
	//	E_BA_AC_OpMod01.eAlarm;
	OuADmpOpMod.arrOpModVal[E_BA_AC_OpMod01.eAlarm]				:= FALSE;
	OuADmpOpMod.arrIgnoreDelayOnVal[E_BA_AC_OpMod01.eAlarm]		:= TRUE;
	OuADmpOpMod.arrIgnoreDelayOffVal[E_BA_AC_OpMod01.eAlarm]		:= FALSE;
	OuADmpOpMod.arrIgnoreFdbVal[E_BA_AC_OpMod01.eAlarm]			:= TRUE;
	//////////////////////////////////////////////
	//////////////////////////////////////////////
	//	E_BA_AC_OpMod01.eForcedVentilation;
	OuADmpOpMod.arrOpModVal[E_BA_AC_OpMod01.eForcedVentilation]				:= TRUE;
	OuADmpOpMod.arrIgnoreDelayOnVal[E_BA_AC_OpMod01.eForcedVentilation]		:= TRUE;
	OuADmpOpMod.arrIgnoreDelayOffVal[E_BA_AC_OpMod01.eForcedVentilation]		:= TRUE;
	OuADmpOpMod.arrIgnoreFdbVal[E_BA_AC_OpMod01.eForcedVentilation]			:= FALSE;
	//////////////////////////////////////////////
	//////////////////////////////////////////////
	//	E_BA_AC_OpMod01.eCentralSwitchOff;
	OuADmpOpMod.arrOpModVal[E_BA_AC_OpMod01.eCentralSwitchOff]				:= FALSE;
	OuADmpOpMod.arrIgnoreDelayOnVal[E_BA_AC_OpMod01.eCentralSwitchOff]		:= TRUE;
	OuADmpOpMod.arrIgnoreDelayOffVal[E_BA_AC_OpMod01.eCentralSwitchOff]		:= FALSE;
	OuADmpOpMod.arrIgnoreFdbVal[E_BA_AC_OpMod01.eCentralSwitchOff]			:= TRUE;
	//////////////////////////////////////////////
	//////////////////////////////////////////////
	//	E_BA_AC_OpMod01.eCustomer01
	OuADmpOpMod.arrOpModVal[E_BA_AC_OpMod01.eCustomer01]				:= FALSE;
	OuADmpOpMod.arrIgnoreDelayOnVal[E_BA_AC_OpMod01.eCustomer01]		:= TRUE;
	OuADmpOpMod.arrIgnoreDelayOffVal[E_BA_AC_OpMod01.eCustomer01]	:= FALSE;
	OuADmpOpMod.arrIgnoreFdbVal[E_BA_AC_OpMod01.eCustomer01]			:= TRUE;
	//////////////////////////////////////////////
	//////////////////////////////////////////////
	//	E_BA_AC_OpMod01.eCustomer02
	OuADmpOpMod.arrOpModVal[E_BA_AC_OpMod01.eCustomer02]				:= FALSE;
	OuADmpOpMod.arrIgnoreDelayOnVal[E_BA_AC_OpMod01.eCustomer02]		:= TRUE;
	OuADmpOpMod.arrIgnoreDelayOffVal[E_BA_AC_OpMod01.eCustomer02]	:= FALSE;
	OuADmpOpMod.arrIgnoreFdbVal[E_BA_AC_OpMod01.eCustomer02]			:= TRUE;
END_IF
END_METHOD

METHOD InitPreHtr
VAR_INPUT
END_VAR
IF	PreHtrOpMod.bInit
THEN	
	PreHtrOpMod.bInit := FALSE;
	//////////////////////////////////////////////
	//////////////////////////////////////////////
	//	E_BA_AC_OpMod01.eOff;
	PreHtrOpMod.arrOpModVal[E_BA_AC_OpMod01.eOff]				:= FALSE;
	PreHtrOpMod.arrIgnoreDelayOnVal[E_BA_AC_OpMod01.eOff]		:= TRUE;
	PreHtrOpMod.arrIgnoreDelayOffVal[E_BA_AC_OpMod01.eOff]		:= TRUE;
	PreHtrOpMod.arrIgnoreFdbVal[E_BA_AC_OpMod01.eOff]			:= TRUE;
	//////////////////////////////////////////////
	//////////////////////////////////////////////
	//	E_BA_AC_OpMod01.eOn;
	PreHtrOpMod.arrOpModVal[E_BA_AC_OpMod01.eOn]				:= TRUE;
	PreHtrOpMod.arrIgnoreDelayOnVal[E_BA_AC_OpMod01.eOn]		:= TRUE;
	PreHtrOpMod.arrIgnoreDelayOffVal[E_BA_AC_OpMod01.eOn]	:= TRUE;
	PreHtrOpMod.arrIgnoreFdbVal[E_BA_AC_OpMod01.eOn]			:= FALSE;
	//////////////////////////////////////////////
	//////////////////////////////////////////////
	//	E_BA_AC_OpMod01.eEmergency;
	PreHtrOpMod.arrOpModVal[E_BA_AC_OpMod01.eEmergency]				:= FALSE;
	PreHtrOpMod.arrIgnoreDelayOnVal[E_BA_AC_OpMod01.eEmergency]		:= TRUE;
	PreHtrOpMod.arrIgnoreDelayOffVal[E_BA_AC_OpMod01.eEmergency]		:= TRUE;
	PreHtrOpMod.arrIgnoreFdbVal[E_BA_AC_OpMod01.eEmergency]			:= TRUE;
	//////////////////////////////////////////////
	//////////////////////////////////////////////
	//	E_BA_AC_OpMod01.eFrost;
	PreHtrOpMod.arrOpModVal[E_BA_AC_OpMod01.eFrost]				:= FALSE;
	PreHtrOpMod.arrIgnoreDelayOnVal[E_BA_AC_OpMod01.eFrost]		:= TRUE;
	PreHtrOpMod.arrIgnoreDelayOffVal[E_BA_AC_OpMod01.eFrost]		:= TRUE;
	PreHtrOpMod.arrIgnoreFdbVal[E_BA_AC_OpMod01.eFrost]			:= TRUE;
	//////////////////////////////////////////////
	//////////////////////////////////////////////
	//	E_BA_AC_OpMod01.eSmokeExtractionProgram;
	PreHtrOpMod.arrOpModVal[E_BA_AC_OpMod01.eSmokeExtractionProgram]				:= TRUE;
	PreHtrOpMod.arrIgnoreDelayOnVal[E_BA_AC_OpMod01.eSmokeExtractionProgram]		:= TRUE;
	PreHtrOpMod.arrIgnoreDelayOffVal[E_BA_AC_OpMod01.eSmokeExtractionProgram]	:= TRUE;
	PreHtrOpMod.arrIgnoreFdbVal[E_BA_AC_OpMod01.eSmokeExtractionProgram]			:= TRUE;
	//////////////////////////////////////////////
	//////////////////////////////////////////////
	//	E_BA_AC_OpMod01.eSmokeExtractionSupplyAir;
	PreHtrOpMod.arrOpModVal[E_BA_AC_OpMod01.eSmokeExtractionSupplyAir]				:= TRUE;
	PreHtrOpMod.arrIgnoreDelayOnVal[E_BA_AC_OpMod01.eSmokeExtractionSupplyAir]		:= TRUE;
	PreHtrOpMod.arrIgnoreDelayOffVal[E_BA_AC_OpMod01.eSmokeExtractionSupplyAir]		:= TRUE;
	PreHtrOpMod.arrIgnoreFdbVal[E_BA_AC_OpMod01.eSmokeExtractionSupplyAir]			:= TRUE;
	//////////////////////////////////////////////
	//////////////////////////////////////////////
	//	E_BA_AC_OpMod01.eSmokeExtractionExhaustAir;
	PreHtrOpMod.arrOpModVal[E_BA_AC_OpMod01.eSmokeExtractionExhaustAir]				:= FALSE;
	PreHtrOpMod.arrIgnoreDelayOnVal[E_BA_AC_OpMod01.eSmokeExtractionExhaustAir]		:= TRUE;
	PreHtrOpMod.arrIgnoreDelayOffVal[E_BA_AC_OpMod01.eSmokeExtractionExhaustAir]		:= TRUE;
	PreHtrOpMod.arrIgnoreFdbVal[E_BA_AC_OpMod01.eSmokeExtractionExhaustAir]			:= TRUE;
	//////////////////////////////////////////////
	//////////////////////////////////////////////
	//	E_BA_AC_OpMod01.eFire;
	PreHtrOpMod.arrOpModVal[E_BA_AC_OpMod01.eFire]				:= FALSE;
	PreHtrOpMod.arrIgnoreDelayOnVal[E_BA_AC_OpMod01.eFire]		:= TRUE;
	PreHtrOpMod.arrIgnoreDelayOffVal[E_BA_AC_OpMod01.eFire]		:= TRUE;
	PreHtrOpMod.arrIgnoreFdbVal[E_BA_AC_OpMod01.eFire]			:= TRUE;
	//////////////////////////////////////////////
	//////////////////////////////////////////////
	//	E_BA_AC_OpMod01.eNightCooling;
	PreHtrOpMod.arrOpModVal[E_BA_AC_OpMod01.eNightCooling]				:= FALSE;
	PreHtrOpMod.arrIgnoreDelayOnVal[E_BA_AC_OpMod01.eNightCooling]		:= TRUE;
	PreHtrOpMod.arrIgnoreDelayOffVal[E_BA_AC_OpMod01.eNightCooling]		:= TRUE;
	PreHtrOpMod.arrIgnoreFdbVal[E_BA_AC_OpMod01.eNightCooling]			:= TRUE;
	//////////////////////////////////////////////
	//////////////////////////////////////////////
	//	E_BA_AC_OpMod01.eCoolDownProtection;
	PreHtrOpMod.arrOpModVal[E_BA_AC_OpMod01.eCoolDownProtection]				:= TRUE;
	PreHtrOpMod.arrIgnoreDelayOnVal[E_BA_AC_OpMod01.eCoolDownProtection]		:= TRUE;
	PreHtrOpMod.arrIgnoreDelayOffVal[E_BA_AC_OpMod01.eCoolDownProtection]	:= TRUE;
	PreHtrOpMod.arrIgnoreFdbVal[E_BA_AC_OpMod01.eCoolDownProtection]			:= FALSE;
	//////////////////////////////////////////////
	//////////////////////////////////////////////
	//	E_BA_AC_OpMod01.eOverHeatingProtection;
	PreHtrOpMod.arrOpModVal[E_BA_AC_OpMod01.eOverHeatingProtection]				:= FALSE;
	PreHtrOpMod.arrIgnoreDelayOnVal[E_BA_AC_OpMod01.eOverHeatingProtection]		:= TRUE;
	PreHtrOpMod.arrIgnoreDelayOffVal[E_BA_AC_OpMod01.eOverHeatingProtection]		:= TRUE;
	PreHtrOpMod.arrIgnoreFdbVal[E_BA_AC_OpMod01.eOverHeatingProtection]			:= TRUE;
	//////////////////////////////////////////////
	//////////////////////////////////////////////
	//	E_BA_AC_OpMod01.eAlarm;
	PreHtrOpMod.arrOpModVal[E_BA_AC_OpMod01.eAlarm]				:= FALSE;
	PreHtrOpMod.arrIgnoreDelayOnVal[E_BA_AC_OpMod01.eAlarm]		:= TRUE;
	PreHtrOpMod.arrIgnoreDelayOffVal[E_BA_AC_OpMod01.eAlarm]		:= TRUE;
	PreHtrOpMod.arrIgnoreFdbVal[E_BA_AC_OpMod01.eAlarm]			:= TRUE;
	//////////////////////////////////////////////
	//////////////////////////////////////////////
	//	E_BA_AC_OpMod01.eForcedVentilation;
	PreHtrOpMod.arrOpModVal[E_BA_AC_OpMod01.eForcedVentilation]				:= TRUE;
	PreHtrOpMod.arrIgnoreDelayOnVal[E_BA_AC_OpMod01.eForcedVentilation]		:= TRUE;
	PreHtrOpMod.arrIgnoreDelayOffVal[E_BA_AC_OpMod01.eForcedVentilation]		:= TRUE;
	PreHtrOpMod.arrIgnoreFdbVal[E_BA_AC_OpMod01.eForcedVentilation]			:= FALSE;
	//////////////////////////////////////////////
	//////////////////////////////////////////////
	//	E_BA_AC_OpMod01.eCentralSwitchOff;
	PreHtrOpMod.arrOpModVal[E_BA_AC_OpMod01.eCentralSwitchOff]				:= FALSE;
	PreHtrOpMod.arrIgnoreDelayOnVal[E_BA_AC_OpMod01.eCentralSwitchOff]		:= TRUE;
	PreHtrOpMod.arrIgnoreDelayOffVal[E_BA_AC_OpMod01.eCentralSwitchOff]		:= TRUE;
	PreHtrOpMod.arrIgnoreFdbVal[E_BA_AC_OpMod01.eCentralSwitchOff]			:= TRUE;
	//////////////////////////////////////////////
	//////////////////////////////////////////////
	//	E_BA_AC_OpMod01.eCustomer01;
	PreHtrOpMod.arrOpModVal[E_BA_AC_OpMod01.eCustomer01]				:= FALSE;
	PreHtrOpMod.arrIgnoreDelayOnVal[E_BA_AC_OpMod01.eCustomer01]		:= TRUE;
	PreHtrOpMod.arrIgnoreDelayOffVal[E_BA_AC_OpMod01.eCustomer01]	:= TRUE;
	PreHtrOpMod.arrIgnoreFdbVal[E_BA_AC_OpMod01.eCustomer01]			:= TRUE;
	//////////////////////////////////////////////
	//////////////////////////////////////////////
	//	E_BA_AC_OpMod01.eCustomer02;
	PreHtrOpMod.arrOpModVal[E_BA_AC_OpMod01.eCustomer02]				:= FALSE;
	PreHtrOpMod.arrIgnoreDelayOnVal[E_BA_AC_OpMod01.eCustomer02]		:= TRUE;
	PreHtrOpMod.arrIgnoreDelayOffVal[E_BA_AC_OpMod01.eCustomer02]	:= TRUE;
	PreHtrOpMod.arrIgnoreFdbVal[E_BA_AC_OpMod01.eCustomer02]			:= TRUE;
END_IF
END_METHOD

METHOD InitSuAFan
VAR_INPUT
END_VAR
IF	SuAFanOpMod.bInit
THEN	
	SuAFanOpMod.bInit := FALSE;
	//////////////////////////////////////////////
	//////////////////////////////////////////////
	//	E_BA_AC_OpMod01.eOff;
	SuAFanOpMod.arrOpModVal[E_BA_AC_OpMod01.eOff]				:= E_BA_Mdlt.eOff;
	SuAFanOpMod.arrIgnoreDelayOnVal[E_BA_AC_OpMod01.eOff]		:= TRUE;
	SuAFanOpMod.arrIgnoreDelayOffVal[E_BA_AC_OpMod01.eOff]		:= TRUE;
	SuAFanOpMod.arrIgnoreFdbVal[E_BA_AC_OpMod01.eOff]			:= TRUE;
	//////////////////////////////////////////////
	//////////////////////////////////////////////
	//	E_BA_AC_OpMod01.eOn;
	SuAFanOpMod.arrOpModVal[E_BA_AC_OpMod01.eOn]				:= E_BA_Mdlt.eOn;
	SuAFanOpMod.arrIgnoreDelayOnVal[E_BA_AC_OpMod01.eOn]		:= TRUE;
	SuAFanOpMod.arrIgnoreDelayOffVal[E_BA_AC_OpMod01.eOn]	:= TRUE;
	SuAFanOpMod.arrIgnoreFdbVal[E_BA_AC_OpMod01.eOn]			:= TRUE;
	//////////////////////////////////////////////
	//////////////////////////////////////////////
	//	E_BA_AC_OpMod01.eEmergency;
	SuAFanOpMod.arrOpModVal[E_BA_AC_OpMod01.eEmergency]				:= E_BA_Mdlt.eOff;
	SuAFanOpMod.arrIgnoreDelayOnVal[E_BA_AC_OpMod01.eEmergency]		:= TRUE;
	SuAFanOpMod.arrIgnoreDelayOffVal[E_BA_AC_OpMod01.eEmergency]		:= TRUE;
	SuAFanOpMod.arrIgnoreFdbVal[E_BA_AC_OpMod01.eEmergency]			:= TRUE;
	//////////////////////////////////////////////
	//////////////////////////////////////////////
	//	E_BA_AC_OpMod01.eFrost;
	SuAFanOpMod.arrOpModVal[E_BA_AC_OpMod01.eFrost]				:= E_BA_Mdlt.eOff;
	SuAFanOpMod.arrIgnoreDelayOnVal[E_BA_AC_OpMod01.eFrost]		:= TRUE;
	SuAFanOpMod.arrIgnoreDelayOffVal[E_BA_AC_OpMod01.eFrost]		:= TRUE;
	SuAFanOpMod.arrIgnoreFdbVal[E_BA_AC_OpMod01.eFrost]			:= TRUE;
	//////////////////////////////////////////////
	//////////////////////////////////////////////
	//	E_BA_AC_OpMod01.eSmokeExtractionProgram;
	SuAFanOpMod.arrOpModVal[E_BA_AC_OpMod01.eSmokeExtractionProgram]				:= E_BA_Mdlt.eOn;
	SuAFanOpMod.arrIgnoreDelayOnVal[E_BA_AC_OpMod01.eSmokeExtractionProgram]		:= TRUE;
	SuAFanOpMod.arrIgnoreDelayOffVal[E_BA_AC_OpMod01.eSmokeExtractionProgram]		:= TRUE;
	SuAFanOpMod.arrIgnoreFdbVal[E_BA_AC_OpMod01.eSmokeExtractionProgram]			:= TRUE;
	//////////////////////////////////////////////
	//////////////////////////////////////////////
	//	E_BA_AC_OpMod01.eSmokeExtractionSupplyAir;
	SuAFanOpMod.arrOpModVal[E_BA_AC_OpMod01.eSmokeExtractionSupplyAir]				:= E_BA_Mdlt.eOn;
	SuAFanOpMod.arrIgnoreDelayOnVal[E_BA_AC_OpMod01.eSmokeExtractionSupplyAir]		:= TRUE;
	SuAFanOpMod.arrIgnoreDelayOffVal[E_BA_AC_OpMod01.eSmokeExtractionSupplyAir]		:= TRUE;
	SuAFanOpMod.arrIgnoreFdbVal[E_BA_AC_OpMod01.eSmokeExtractionSupplyAir]			:= TRUE;
	//////////////////////////////////////////////
	//////////////////////////////////////////////
	//	E_BA_AC_OpMod01.eSmokeExtractionExhaustAir;
	SuAFanOpMod.arrOpModVal[E_BA_AC_OpMod01.eSmokeExtractionExhaustAir]				:= E_BA_Mdlt.eOff;
	SuAFanOpMod.arrIgnoreDelayOnVal[E_BA_AC_OpMod01.eSmokeExtractionExhaustAir]		:= TRUE;
	SuAFanOpMod.arrIgnoreDelayOffVal[E_BA_AC_OpMod01.eSmokeExtractionExhaustAir]		:= TRUE;
	SuAFanOpMod.arrIgnoreFdbVal[E_BA_AC_OpMod01.eSmokeExtractionExhaustAir]			:= TRUE;
	//////////////////////////////////////////////
	//////////////////////////////////////////////
	//	E_BA_AC_OpMod01.eFire;
	SuAFanOpMod.arrOpModVal[E_BA_AC_OpMod01.eFire]				:= E_BA_Mdlt.eOff;
	SuAFanOpMod.arrIgnoreDelayOnVal[E_BA_AC_OpMod01.eFire]		:= TRUE;
	SuAFanOpMod.arrIgnoreDelayOffVal[E_BA_AC_OpMod01.eFire]		:= TRUE;
	SuAFanOpMod.arrIgnoreFdbVal[E_BA_AC_OpMod01.eFire]			:= TRUE;
	//////////////////////////////////////////////
	//////////////////////////////////////////////
	//	E_BA_AC_OpMod01.eNightCooling;
	SuAFanOpMod.arrOpModVal[E_BA_AC_OpMod01.eNightCooling]				:= E_BA_Mdlt.eOn;
	SuAFanOpMod.arrIgnoreDelayOnVal[E_BA_AC_OpMod01.eNightCooling]		:= TRUE;
	SuAFanOpMod.arrIgnoreDelayOffVal[E_BA_AC_OpMod01.eNightCooling]		:= TRUE;
	SuAFanOpMod.arrIgnoreFdbVal[E_BA_AC_OpMod01.eNightCooling]			:= TRUE;
	//////////////////////////////////////////////
	//////////////////////////////////////////////
	//	E_BA_AC_OpMod01.eCoolDownProtection;
	SuAFanOpMod.arrOpModVal[E_BA_AC_OpMod01.eCoolDownProtection]				:= E_BA_Mdlt.eOn;
	SuAFanOpMod.arrIgnoreDelayOnVal[E_BA_AC_OpMod01.eCoolDownProtection]		:= TRUE;
	SuAFanOpMod.arrIgnoreDelayOffVal[E_BA_AC_OpMod01.eCoolDownProtection]	:= TRUE;
	SuAFanOpMod.arrIgnoreFdbVal[E_BA_AC_OpMod01.eCoolDownProtection]			:= TRUE;
	//////////////////////////////////////////////
	//////////////////////////////////////////////
	//	E_BA_AC_OpMod01.eOverHeatingProtection;
	SuAFanOpMod.arrOpModVal[E_BA_AC_OpMod01.eOverHeatingProtection]				:= E_BA_Mdlt.eOn;
	SuAFanOpMod.arrIgnoreDelayOnVal[E_BA_AC_OpMod01.eOverHeatingProtection]		:= TRUE;
	SuAFanOpMod.arrIgnoreDelayOffVal[E_BA_AC_OpMod01.eOverHeatingProtection]		:= TRUE;
	SuAFanOpMod.arrIgnoreFdbVal[E_BA_AC_OpMod01.eOverHeatingProtection]			:= TRUE;
	//////////////////////////////////////////////
	//////////////////////////////////////////////
	//	E_BA_AC_OpMod01.eAlarm;
	SuAFanOpMod.arrOpModVal[E_BA_AC_OpMod01.eAlarm]				:= E_BA_Mdlt.eOff;
	SuAFanOpMod.arrIgnoreDelayOnVal[E_BA_AC_OpMod01.eAlarm]		:= TRUE;
	SuAFanOpMod.arrIgnoreDelayOffVal[E_BA_AC_OpMod01.eAlarm]		:= TRUE;
	SuAFanOpMod.arrIgnoreFdbVal[E_BA_AC_OpMod01.eAlarm]			:= TRUE;
	//////////////////////////////////////////////
	//////////////////////////////////////////////
	//	E_BA_AC_OpMod01.eForcedVentilation;
	SuAFanOpMod.arrOpModVal[E_BA_AC_OpMod01.eForcedVentilation]				:= E_BA_Mdlt.eOn;
	SuAFanOpMod.arrIgnoreDelayOnVal[E_BA_AC_OpMod01.eForcedVentilation]		:= TRUE;
	SuAFanOpMod.arrIgnoreDelayOffVal[E_BA_AC_OpMod01.eForcedVentilation]		:= TRUE;
	SuAFanOpMod.arrIgnoreFdbVal[E_BA_AC_OpMod01.eForcedVentilation]			:= TRUE;
	//////////////////////////////////////////////
	//////////////////////////////////////////////
	//	E_BA_AC_OpMod01.eCentralSwitchOff;
	SuAFanOpMod.arrOpModVal[E_BA_AC_OpMod01.eCentralSwitchOff]				:= E_BA_Mdlt.eOff;
	SuAFanOpMod.arrIgnoreDelayOnVal[E_BA_AC_OpMod01.eCentralSwitchOff]		:= TRUE;
	SuAFanOpMod.arrIgnoreDelayOffVal[E_BA_AC_OpMod01.eCentralSwitchOff]		:= TRUE;
	SuAFanOpMod.arrIgnoreFdbVal[E_BA_AC_OpMod01.eCentralSwitchOff]			:= TRUE;
	//////////////////////////////////////////////
	//////////////////////////////////////////////
	//	E_BA_AC_OpMod01.eCustomer01;
	SuAFanOpMod.arrOpModVal[E_BA_AC_OpMod01.eCustomer01]				:= E_BA_Mdlt.eOff;
	SuAFanOpMod.arrIgnoreDelayOnVal[E_BA_AC_OpMod01.eCustomer01]		:= TRUE;
	SuAFanOpMod.arrIgnoreDelayOffVal[E_BA_AC_OpMod01.eCustomer01]	:= TRUE;
	SuAFanOpMod.arrIgnoreFdbVal[E_BA_AC_OpMod01.eCustomer01]			:= TRUE;
	//////////////////////////////////////////////
	//////////////////////////////////////////////
	//	E_BA_AC_OpMod01.eCustomer02;
	SuAFanOpMod.arrOpModVal[E_BA_AC_OpMod01.eCustomer02]				:= E_BA_Mdlt.eOff;
	SuAFanOpMod.arrIgnoreDelayOnVal[E_BA_AC_OpMod01.eCustomer02]		:= TRUE;
	SuAFanOpMod.arrIgnoreDelayOffVal[E_BA_AC_OpMod01.eCustomer02]	:= TRUE;
	SuAFanOpMod.arrIgnoreFdbVal[E_BA_AC_OpMod01.eCustomer02]			:= TRUE;
END_IF
END_METHOD

METHOD InitTempCtrl
VAR_INPUT
END_VAR
IF	TempCtrlOpMod.bInit
THEN	
	TempCtrlOpMod.bInit := FALSE;
	//////////////////////////////////////////////
	//////////////////////////////////////////////
	//	E_BA_AC_OpMod01.eOff;
	TempCtrlOpMod.arrOpModVal[E_BA_AC_OpMod01.eOff]					:= E_BA_Mdlt.eOff;
	TempCtrlOpMod.arrIgnoreDelayOnVal[E_BA_AC_OpMod01.eOff]			:= TRUE;
	TempCtrlOpMod.arrIgnoreDelayOffVal[E_BA_AC_OpMod01.eOff]			:= TRUE;
	TempCtrlOpMod.arrIgnoreFdbVal[E_BA_AC_OpMod01.eOff]				:= TRUE;
	//////////////////////////////////////////////
	//////////////////////////////////////////////
	//	E_BA_AC_OpMod01.eOn;
	TempCtrlOpMod.arrOpModVal[E_BA_AC_OpMod01.eOn]					:= E_BA_Mdlt.eOn;
	TempCtrlOpMod.arrIgnoreDelayOnVal[E_BA_AC_OpMod01.eOn]			:= FALSE;
	TempCtrlOpMod.arrIgnoreDelayOffVal[E_BA_AC_OpMod01.eOn]			:= TRUE;
	TempCtrlOpMod.arrIgnoreFdbVal[E_BA_AC_OpMod01.eOn]				:= TRUE;
	//////////////////////////////////////////////
	//////////////////////////////////////////////
	//	E_BA_AC_OpMod01.eEmergency;	
	TempCtrlOpMod.arrOpModVal[E_BA_AC_OpMod01.eEmergency]					:= E_BA_Mdlt.eOff;
	TempCtrlOpMod.arrIgnoreDelayOnVal[E_BA_AC_OpMod01.eEmergency]			:= TRUE;
	TempCtrlOpMod.arrIgnoreDelayOffVal[E_BA_AC_OpMod01.eEmergency]			:= TRUE;
	TempCtrlOpMod.arrIgnoreFdbVal[E_BA_AC_OpMod01.eEmergency]				:= TRUE;
	//////////////////////////////////////////////
	//////////////////////////////////////////////
	//	E_BA_AC_OpMod01.eFrost;
	TempCtrlOpMod.arrOpModVal[E_BA_AC_OpMod01.eFrost]					:= E_BA_Mdlt.eOff;
	TempCtrlOpMod.arrIgnoreDelayOnVal[E_BA_AC_OpMod01.eFrost]			:= TRUE;
	TempCtrlOpMod.arrIgnoreDelayOffVal[E_BA_AC_OpMod01.eFrost]			:= TRUE;
	TempCtrlOpMod.arrIgnoreFdbVal[E_BA_AC_OpMod01.eFrost]				:= TRUE;
	//////////////////////////////////////////////
	//////////////////////////////////////////////
	//	E_BA_AC_OpMod01.eSmokeExtractionProgram;
	TempCtrlOpMod.arrOpModVal[E_BA_AC_OpMod01.eSmokeExtractionProgram]					:= E_BA_Mdlt.eOn;
	TempCtrlOpMod.arrIgnoreDelayOnVal[E_BA_AC_OpMod01.eSmokeExtractionProgram]			:= TRUE;
	TempCtrlOpMod.arrIgnoreDelayOffVal[E_BA_AC_OpMod01.eSmokeExtractionProgram]			:= TRUE;
	TempCtrlOpMod.arrIgnoreFdbVal[E_BA_AC_OpMod01.eSmokeExtractionProgram]				:= TRUE;
	//////////////////////////////////////////////
	//////////////////////////////////////////////
	//	E_BA_AC_OpMod01.eSmokeExtractionSupplyAir;
	TempCtrlOpMod.arrOpModVal[E_BA_AC_OpMod01.eSmokeExtractionSupplyAir]					:= E_BA_Mdlt.eOn; 
	TempCtrlOpMod.arrIgnoreDelayOnVal[E_BA_AC_OpMod01.eSmokeExtractionSupplyAir]			:= TRUE; 
	TempCtrlOpMod.arrIgnoreDelayOffVal[E_BA_AC_OpMod01.eSmokeExtractionSupplyAir]			:= TRUE; 
	TempCtrlOpMod.arrIgnoreFdbVal[E_BA_AC_OpMod01.eSmokeExtractionSupplyAir]				:= TRUE; 
	//////////////////////////////////////////////
	//////////////////////////////////////////////
	//	E_BA_AC_OpMod01.eSmokeExtractionExhaustAir;
	TempCtrlOpMod.arrOpModVal[E_BA_AC_OpMod01.eSmokeExtractionExhaustAir]					:= E_BA_Mdlt.eOn; 
	TempCtrlOpMod.arrIgnoreDelayOnVal[E_BA_AC_OpMod01.eSmokeExtractionExhaustAir]			:= TRUE; 
	TempCtrlOpMod.arrIgnoreDelayOffVal[E_BA_AC_OpMod01.eSmokeExtractionExhaustAir]			:= TRUE; 
	TempCtrlOpMod.arrIgnoreFdbVal[E_BA_AC_OpMod01.eSmokeExtractionExhaustAir]				:= TRUE; 
	//////////////////////////////////////////////
	//////////////////////////////////////////////
	//	E_BA_AC_OpMod01.eFire;
	TempCtrlOpMod.arrOpModVal[E_BA_AC_OpMod01.eFire]					:= E_BA_Mdlt.eOff; 
	TempCtrlOpMod.arrIgnoreDelayOnVal[E_BA_AC_OpMod01.eFire]			:= TRUE; 
	TempCtrlOpMod.arrIgnoreDelayOffVal[E_BA_AC_OpMod01.eFire]			:= TRUE; 
	TempCtrlOpMod.arrIgnoreFdbVal[E_BA_AC_OpMod01.eFire]				:= TRUE; 
	//////////////////////////////////////////////
	//////////////////////////////////////////////
	//	E_BA_AC_OpMod01.eNightCooling;
	TempCtrlOpMod.arrOpModVal[E_BA_AC_OpMod01.eNightCooling]					:= E_BA_Mdlt.eOn; 
	TempCtrlOpMod.arrIgnoreDelayOnVal[E_BA_AC_OpMod01.eNightCooling]			:= FALSE; 
	TempCtrlOpMod.arrIgnoreDelayOffVal[E_BA_AC_OpMod01.eNightCooling]			:= TRUE; 
	TempCtrlOpMod.arrIgnoreFdbVal[E_BA_AC_OpMod01.eNightCooling]				:= TRUE; 
	//////////////////////////////////////////////
	//////////////////////////////////////////////
	//	E_BA_AC_OpMod01.eCoolDownProtection;
	TempCtrlOpMod.arrOpModVal[E_BA_AC_OpMod01.eCoolDownProtection]				:= E_BA_Mdlt.eMax; 
	TempCtrlOpMod.arrIgnoreDelayOnVal[E_BA_AC_OpMod01.eCoolDownProtection]		:= FALSE; 
	TempCtrlOpMod.arrIgnoreDelayOffVal[E_BA_AC_OpMod01.eCoolDownProtection]		:= TRUE; 
	TempCtrlOpMod.arrIgnoreFdbVal[E_BA_AC_OpMod01.eCoolDownProtection]			:= TRUE; 
	//////////////////////////////////////////////
	//////////////////////////////////////////////
	//	E_BA_AC_OpMod01.eOverHeatingProtection;
	TempCtrlOpMod.arrOpModVal[E_BA_AC_OpMod01.eOverHeatingProtection]				:= E_BA_Mdlt.eOn; 
	TempCtrlOpMod.arrIgnoreDelayOnVal[E_BA_AC_OpMod01.eOverHeatingProtection]		:= FALSE; 
	TempCtrlOpMod.arrIgnoreDelayOffVal[E_BA_AC_OpMod01.eOverHeatingProtection]		:= TRUE; 
	TempCtrlOpMod.arrIgnoreFdbVal[E_BA_AC_OpMod01.eOverHeatingProtection]			:= TRUE; 
	//////////////////////////////////////////////
	//////////////////////////////////////////////
	//	E_BA_AC_OpMod01.eAlarm;
	TempCtrlOpMod.arrOpModVal[E_BA_AC_OpMod01.eAlarm]				:= E_BA_Mdlt.eOff;
	TempCtrlOpMod.arrIgnoreDelayOnVal[E_BA_AC_OpMod01.eAlarm]		:= TRUE;
	TempCtrlOpMod.arrIgnoreDelayOffVal[E_BA_AC_OpMod01.eAlarm]		:= TRUE;
	TempCtrlOpMod.arrIgnoreFdbVal[E_BA_AC_OpMod01.eAlarm]			:= TRUE;
	//////////////////////////////////////////////
	//////////////////////////////////////////////
	//	E_BA_AC_OpMod01.eForcedVentilation;
	TempCtrlOpMod.arrOpModVal[E_BA_AC_OpMod01.eForcedVentilation]				:= E_BA_Mdlt.eOn;
	TempCtrlOpMod.arrIgnoreDelayOnVal[E_BA_AC_OpMod01.eForcedVentilation]		:= FALSE;
	TempCtrlOpMod.arrIgnoreDelayOffVal[E_BA_AC_OpMod01.eForcedVentilation]		:= TRUE;
	TempCtrlOpMod.arrIgnoreFdbVal[E_BA_AC_OpMod01.eForcedVentilation]			:= TRUE;
	//////////////////////////////////////////////
	//////////////////////////////////////////////
	//	E_BA_AC_OpMod01.eCentralSwitchOff;  	
	TempCtrlOpMod.arrOpModVal[E_BA_AC_OpMod01.eCentralSwitchOff]				:= E_BA_Mdlt.eOff;
	TempCtrlOpMod.arrIgnoreDelayOnVal[E_BA_AC_OpMod01.eCentralSwitchOff]		:= TRUE;
	TempCtrlOpMod.arrIgnoreDelayOffVal[E_BA_AC_OpMod01.eCentralSwitchOff]		:= TRUE;
	TempCtrlOpMod.arrIgnoreFdbVal[E_BA_AC_OpMod01.eCentralSwitchOff]			:= TRUE;
	//////////////////////////////////////////////
	//////////////////////////////////////////////
	//	E_BA_AC_OpMod01.eCustomer01
	TempCtrlOpMod.arrOpModVal[E_BA_AC_OpMod01.eCustomer01]				:= E_BA_Mdlt.eOff;
	TempCtrlOpMod.arrIgnoreDelayOnVal[E_BA_AC_OpMod01.eCustomer01]		:= TRUE;
	TempCtrlOpMod.arrIgnoreDelayOffVal[E_BA_AC_OpMod01.eCustomer01]		:= TRUE;
	TempCtrlOpMod.arrIgnoreFdbVal[E_BA_AC_OpMod01.eCustomer01]			:= TRUE;
	//////////////////////////////////////////////
	//////////////////////////////////////////////
	//	E_BA_AC_OpMod01.eCustomer02          	
	TempCtrlOpMod.arrOpModVal[E_BA_AC_OpMod01.eCustomer02]				:= E_BA_Mdlt.eOff;
	TempCtrlOpMod.arrIgnoreDelayOnVal[E_BA_AC_OpMod01.eCustomer02]		:= TRUE;
	TempCtrlOpMod.arrIgnoreDelayOffVal[E_BA_AC_OpMod01.eCustomer02]		:= TRUE;
	TempCtrlOpMod.arrIgnoreFdbVal[E_BA_AC_OpMod01.eCustomer02]			:= TRUE;
END_IF
END_METHOD

END_FUNCTION_BLOCK

// ---- Templates/POUs/Trade/AirConditioning/General/FB_BA_AC_SeqT.TcPOU
{region '#Template'}
	{attribute 'Version' := '5.0.2.0'}
	{attribute 'Tags' := '"LCID": "1031", "Text": "AC, Allgemein, AHU, Sequenz, Sequenzverbindung, Temperatur"'}
	{attribute 'Tags' := '"LCID": "1033", "Text": "AC, General, AHU, Sequence, Sequence link, Temperature"'}
	{attribute 'Using' := '"Type": "Template", "URI": "E_BA_AC_OpMod01"'}
	{attribute 'Using' := '"Type": "Template", "URI": "E_BA_AC_SeqNumber_T"'}
	{attribute 'Description' := '"LCID": "1031", "Text": "Sequenzverbindung"'}
	{attribute 'Description' := '"LCID": "1033", "Text": "Sequence link"'}
{endregion}

FUNCTION_BLOCK FB_BA_AC_SeqT EXTENDS FB_BA_View
VAR_INPUT
	bEn					: BOOL;
	eOpMode				: E_BA_AC_OpMod01;		
	fTWth				: REAL;
END_VAR
VAR_OUTPUT
	bSumLmt				: BOOL;		//Sommer Grenzwert ist aktiv	//	Summer limit is active
	bWinLmt				: BOOL;		//Winter Grenzwert ist aktiv	//	Winter limit is active
	nActvSeqCtrl		: UDINT;	// Nummer des aktiven Sequenzcontrollers // number of the active sequenz controller
END_VAR
VAR_IN_OUT
	stTSeqLink			: ST_BA_SeqLink;	//	Sequenz Link Struktur	//	Sequence link structure	
END_VAR
VAR_INPUT CONSTANT
	WthTLmtSum			: FB_BA_AV_Op;
	WthTLmtWin			: FB_BA_AV_Op;
	SeqLink				: FB_BA_SequenceLinkBase;		//	Hauptprogramm zur Steuerung der Sequenzregler einer Anlage	//	Main program to control the sequence controller of a plant
	ActvSeqCtrl			: FB_BA_MV_Op;	
END_VAR
VAR
	WthTLmtWinHys		: FB_BA_Swi2P;			//	Hysterese Grenzwert Winter									//	Hysteresis limit winter
	WthTLmtSumHys		: FB_BA_Swi2P;			//	Hysterese Grenzwert Sommer									//	Hysteresis limit summer
	StartSeq			: FB_BA_PrioSwi_UDI08;	//	Festlegung Start Sequenz									//	Fixing start-up sequence
END_VAR

SUPER^(); // FB_BA_View
WthTLmtSum(); // FB_BA_AV_Op
WthTLmtWin(); // FB_BA_AV_Op
WthTLmtWinHys(
    bEn := TRUE,
    fIn := fTWth,
    fOn := WthTLmtWin.fPresentValue,
    fOff := WthTLmtWin.fPresentValue + 1); // FB_BA_Swi2P
bWinLmt := WthTLmtWinHys.bQ;
WthTLmtSumHys(
    bEn := TRUE,
    fIn := fTWth,
    fOn := WthTLmtSum.fPresentValue,
    fOff := WthTLmtSum.fPresentValue - 1); // FB_BA_Swi2P
bSumLmt := WthTLmtSumHys.bQ;
StartSeq(
    bEn01 := eOpMode = E_BA_AC_OpMod01.eOverHeatingProtection,
    nVal01 := E_BA_AC_SeqNumber_T.eCooler,
    bEn02 := eOpMode = E_BA_AC_OpMod01.eCoolDownProtection,
    nVal02 := E_BA_AC_SeqNumber_T.ePreHeater,
    bEn04 := bWinLmt,
    nVal04 := E_BA_AC_SeqNumber_T.ePreHeater,
    bEn05 := bSumLmt,
    nVal05 := E_BA_AC_SeqNumber_T.eCooler,
    bEn08 := TRUE,
    nVal08 := E_BA_AC_SeqNumber_T.eEnergyRecovery); // FB_BA_PrioSwi_UDI08
SeqLink(bEn := bEn, nNumStartCtrl := StartSeq.nVal, nSwiOverTi := 10, stSeqLink := stTSeqLink); // FB_BA_SequenceLinkBase
ActvSeqCtrl(nValuePgm := SEL(SeqLink.nActvSeqCtrl > 0, E_BA_AC_SeqNumber_T.eOff, SeqLink.nActvSeqCtrl)); // FB_BA_MV_Op
nActvSeqCtrl := ActvSeqCtrl.nPresentValue;

METHOD FB_init : BOOL
VAR_INPUT
	bInitRetains : BOOL; // if TRUE, the retain variables are initialized (warm start / cold start)
	bInCopyCode : BOOL;  // if TRUE, the instance afterwards gets moved into the copy code (online change)
END_VAR
WthTLmtSum.iParent							:= THIS^;
WthTLmtSum.iLabel							:= LblCtl_LimitValueWeatherTemperatureSummer;
WthTLmtSum.eUnit 							:= E_BA_Unit.eTemperature_DegreesCelsius;								 
WthTLmtSum.fValueRm							:= 10;	
WthTLmtSum.fCOVIncrement					:= BA2_Param.fDefCOVIncrement;		

WthTLmtWin.iParent							:= THIS^;
WthTLmtWin.iLabel							:= LblCtl_LimitValueWeatherTemperatureWinter;
WthTLmtWin.eUnit 							:= E_BA_Unit.eTemperature_DegreesCelsius;								 
WthTLmtWin.fValueRm							:= 20;	
WthTLmtWin.fCOVIncrement					:= BA2_Param.fDefCOVIncrement;		

SeqLink.fHys								:= 2;
SeqLink.eNoStartCtrlFound					:= E_BA_NoStartCtrlFound.eLastActionReverse;	
SeqLink.eNoEnableSeqCtrl					:= E_BA_NoEnableSeqCtrl.eNextAction;	

ActvSeqCtrl.iParent							:= THIS^;
ActvSeqCtrl.iLabel							:= LblCtl_CurrentSequenceTemperature;
ActvSeqCtrl.aStateText[1]					:= txtEvent_Reheater;
ActvSeqCtrl.aStateText[2]					:= txtEvent_Preheater;
ActvSeqCtrl.aStateText[3]					:= txtEvent_MixedAir;
ActvSeqCtrl.aStateText[4]					:= txtEvent_EnergyRecovery;
ActvSeqCtrl.aStateText[5]					:= txtEvent_Cooler;
ActvSeqCtrl.aStateText[6]					:= txtEvent_Off;
END_METHOD

END_FUNCTION_BLOCK

// ---- Templates/POUs/Trade/AirConditioning/General/FB_BA_AC_SumNgtCol.TcPOU
{region '#Template'}
	{attribute 'Version' := '5.0.0.0'}
	{attribute 'Tags' := '"LCID": "1031", "Text": "AC, Allgemein, AHU, Nachtkühlung"'}
	{attribute 'Tags' := '"LCID": "1033", "Text": "AC, General, AHU, night cooling"'}
	{attribute 'Using' := '"Type": "Template", "URI": "E_BA_OnOff"'}
	{attribute 'Description' := '"LCID": "1031", "Text": "Nachtkühlung"'}
	{attribute 'Description' := '"LCID": "1033", "Text": "night cooling"'}
{endregion}
FUNCTION_BLOCK FB_BA_AC_SumNgtCol EXTENDS FB_BA_View
VAR_INPUT
	fTRm					: REAL;
	fSpRm					: REAL;
	fTWth					: REAL;		
END_VAR
VAR_OUTPUT
	bQ						: BOOL;
END_VAR
VAR_INPUT CONSTANT
	WthTLoLmt				: FB_BA_AV_Op;	
	RmTHys					: FB_BA_AV_Op;	
	SwiOnDiffT				: FB_BA_AV_Op;	
	SwiOffDiffT				: FB_BA_AV_Op;	
	Q						: FB_BA_BV_Op;																					
	Sched					: FB_BA_SchedM;
END_VAR
VAR
	NgtColFnct				: FB_BA_NgtCol;
END_VAR

SUPER^(); // FB_BA_View
Sched(); // FB_BA_SchedM
WthTLoLmt(); // FB_BA_AV_Op
RmTHys(); // FB_BA_AV_Op
SwiOnDiffT(); // FB_BA_AV_Op
SwiOffDiffT(); // FB_BA_AV_Op
NgtColFnct(
    bEn := Sched.nPresentValue = E_BA_OnOff.eOn,
    fTOts := fTWth,
    fTRm := fTRm,
    fSpRm := fSpRm,
    fTOtsLoLmt := WthTLoLmt.fPresentValue,
    fTRmHys := RmTHys.fPresentValue,
    fSwiOnDiffT := SwiOnDiffT.fPresentValue,
    fSwiOffDiffT := SwiOffDiffT.fPresentValue); // FB_BA_NgtCol
Q(bValuePgm := NgtColFnct.bQ); // FB_BA_BV_Op
bQ := Q.bPresentValue;

METHOD FB_init : BOOL
VAR_INPUT
	bInitRetains : BOOL; // if TRUE, the retain variables are initialized (warm start / cold start)
	bInCopyCode : BOOL;  // if TRUE, the instance afterwards gets moved into the copy code (online change)
END_VAR
WthTLoLmt.iParent			:= THIS^;
WthTLoLmt.iLabel			:= LblCtl_OutsideTemperatureLowLimit; 					
WthTLoLmt.eUnit				:= E_BA_Unit.eTemperature_DegreesCelsius;  
WthTLoLmt.fValueRm			:= 9.0;

RmTHys.iParent				:= THIS^;
RmTHys.iLabel				:= LblCtl_HysteresisRoomTemperature; 									 	 
RmTHys.eUnit				:= E_BA_Unit.eTemperature_DegreesCelsius;  
RmTHys.fValueRm				:= 2.0;

SwiOnDiffT.iParent			:= THIS^; 
SwiOnDiffT.iLabel			:= LblCtl_OnValueDifferenceOutsideInsightTemperature; 									 	 					 	 
SwiOnDiffT.eUnit			:= E_BA_Unit.eTemperature_DegreesCelsius;  
SwiOnDiffT.fValueRm			:= 7.0;

SwiOffDiffT.iParent			:= THIS^; 
SwiOffDiffT.iLabel			:= LblCtl_OffValueDifferenceOutsideInsightTemperature; 								 	 
SwiOffDiffT.eUnit			:= E_BA_Unit.eTemperature_DegreesCelsius;  
SwiOffDiffT.fValueRm		:= 5.0;

Q.iParent					:= THIS^;
Q.iLabel					:= LblFun_OperationalMessage; 			
Q.sInactiveText				:= txtEvent_Off;
Q.sActiveText				:= txtEvent_On;
Q.bValueRm					:= FALSE;								
Q.eToggleMode 				:= E_BA_ToggleMode.eSwitch;

Sched.iParent											:= THIS^;
Sched.iLabel											:= LblFun_Scheduler; 				
Sched.aStateText[1]										:= txtEvent_Off;
Sched.aStateText[2]										:= txtEvent_On;
Sched.nPredictTime										:= 0;
Sched.nDefaultValue										:= E_BA_OnOff.eOff;
Sched.bWriteWeekly										:= FALSE;
//	Monday
Sched.aWeek[E_BA_Weekday.eMonday,1].eState				:= E_BA_SchedEntryState.eValue;
Sched.aWeek[E_BA_Weekday.eMonday,1].uValue.udiVal		:= E_BA_OnOff.eOn;
Sched.aWeek[E_BA_Weekday.eMonday,1].stTime.nHour		:= 1;
Sched.aWeek[E_BA_Weekday.eMonday,1].stTime.nMinute		:= 0;
Sched.aWeek[E_BA_Weekday.eMonday,1].stTime.nSecond		:= 0;
Sched.aWeek[E_BA_Weekday.eMonday,2].eState				:= E_BA_SchedEntryState.eValue;
Sched.aWeek[E_BA_Weekday.eMonday,2].uValue.udiVal		:= E_BA_OnOff.eOff;
Sched.aWeek[E_BA_Weekday.eMonday,2].stTime.nHour		:= 5;
Sched.aWeek[E_BA_Weekday.eMonday,2].stTime.nMinute		:= 0;
Sched.aWeek[E_BA_Weekday.eMonday,2].stTime.nSecond		:= 0;
Sched.aWeek[E_BA_Weekday.eMonday,3].eState				:= E_BA_SchedEntryState.eValue;
Sched.aWeek[E_BA_Weekday.eMonday,3].uValue.udiVal		:= E_BA_OnOff.eOff;
Sched.aWeek[E_BA_Weekday.eMonday,3].stTime.nHour		:= 0;
Sched.aWeek[E_BA_Weekday.eMonday,3].stTime.nMinute		:= 0;
Sched.aWeek[E_BA_Weekday.eMonday,3].stTime.nSecond		:= 0;
//	Tuesday
Sched.aWeek[E_BA_Weekday.eTuesday,1].eState				:= E_BA_SchedEntryState.eValue;
Sched.aWeek[E_BA_Weekday.eTuesday,1].uValue.udiVal		:= E_BA_OnOff.eOn;
Sched.aWeek[E_BA_Weekday.eTuesday,1].stTime.nHour		:= 1;
Sched.aWeek[E_BA_Weekday.eTuesday,1].stTime.nMinute		:= 0;
Sched.aWeek[E_BA_Weekday.eTuesday,1].stTime.nSecond		:= 0;
Sched.aWeek[E_BA_Weekday.eTuesday,2].eState				:= E_BA_SchedEntryState.eValue;
Sched.aWeek[E_BA_Weekday.eTuesday,2].uValue.udiVal		:= E_BA_OnOff.eOff;
Sched.aWeek[E_BA_Weekday.eTuesday,2].stTime.nHour		:= 5;
Sched.aWeek[E_BA_Weekday.eTuesday,2].stTime.nMinute		:= 0;
Sched.aWeek[E_BA_Weekday.eTuesday,2].stTime.nSecond		:= 0;
Sched.aWeek[E_BA_Weekday.eTuesday,3].eState				:= E_BA_SchedEntryState.eValue;
Sched.aWeek[E_BA_Weekday.eTuesday,3].uValue.udiVal		:= E_BA_OnOff.eOff;
Sched.aWeek[E_BA_Weekday.eTuesday,3].stTime.nHour		:= 0;
Sched.aWeek[E_BA_Weekday.eTuesday,3].stTime.nMinute		:= 0;
Sched.aWeek[E_BA_Weekday.eTuesday,3].stTime.nSecond		:= 0;
//	Wednesday
Sched.aWeek[E_BA_Weekday.eWednesday,1].eState			:= E_BA_SchedEntryState.eValue;
Sched.aWeek[E_BA_Weekday.eWednesday,1].uValue.udiVal	:= E_BA_OnOff.eOn;
Sched.aWeek[E_BA_Weekday.eWednesday,1].stTime.nHour		:= 1;
Sched.aWeek[E_BA_Weekday.eWednesday,1].stTime.nMinute	:= 0;
Sched.aWeek[E_BA_Weekday.eWednesday,1].stTime.nSecond	:= 0;
Sched.aWeek[E_BA_Weekday.eWednesday,2].eState			:= E_BA_SchedEntryState.eValue;
Sched.aWeek[E_BA_Weekday.eWednesday,2].uValue.udiVal	:= E_BA_OnOff.eOff;
Sched.aWeek[E_BA_Weekday.eWednesday,2].stTime.nHour		:= 5;
Sched.aWeek[E_BA_Weekday.eWednesday,2].stTime.nMinute	:= 0;
Sched.aWeek[E_BA_Weekday.eWednesday,2].stTime.nSecond	:= 0;
Sched.aWeek[E_BA_Weekday.eWednesday,3].eState			:= E_BA_SchedEntryState.eValue;
Sched.aWeek[E_BA_Weekday.eWednesday,3].uValue.udiVal	:= E_BA_OnOff.eOff;
Sched.aWeek[E_BA_Weekday.eWednesday,3].stTime.nHour		:= 0;
Sched.aWeek[E_BA_Weekday.eWednesday,3].stTime.nMinute	:= 0;
Sched.aWeek[E_BA_Weekday.eWednesday,3].stTime.nSecond	:= 0;
//	Thursday
Sched.aWeek[E_BA_Weekday.eThursday,1].eState			:= E_BA_SchedEntryState.eValue;
Sched.aWeek[E_BA_Weekday.eThursday,1].uValue.udiVal		:= E_BA_OnOff.eOn;
Sched.aWeek[E_BA_Weekday.eThursday,1].stTime.nHour		:= 1;
Sched.aWeek[E_BA_Weekday.eThursday,1].stTime.nMinute	:= 0;
Sched.aWeek[E_BA_Weekday.eThursday,1].stTime.nSecond	:= 0;
Sched.aWeek[E_BA_Weekday.eThursday,2].eState			:= E_BA_SchedEntryState.eValue;
Sched.aWeek[E_BA_Weekday.eThursday,2].uValue.udiVal		:= E_BA_OnOff.eOff;
Sched.aWeek[E_BA_Weekday.eThursday,2].stTime.nHour		:= 5;
Sched.aWeek[E_BA_Weekday.eThursday,2].stTime.nMinute	:= 0;
Sched.aWeek[E_BA_Weekday.eThursday,2].stTime.nSecond	:= 0;
Sched.aWeek[E_BA_Weekday.eThursday,3].eState			:= E_BA_SchedEntryState.eValue;
Sched.aWeek[E_BA_Weekday.eThursday,3].uValue.udiVal		:= E_BA_OnOff.eOff;
Sched.aWeek[E_BA_Weekday.eThursday,3].stTime.nHour		:= 0;
Sched.aWeek[E_BA_Weekday.eThursday,3].stTime.nMinute	:= 0;
Sched.aWeek[E_BA_Weekday.eThursday,3].stTime.nSecond	:= 0;
//	Friday
Sched.aWeek[E_BA_Weekday.eFriday,1].eState				:= E_BA_SchedEntryState.eValue;
Sched.aWeek[E_BA_Weekday.eFriday,1].uValue.udiVal		:= E_BA_OnOff.eOn;
Sched.aWeek[E_BA_Weekday.eFriday,1].stTime.nHour		:= 1;
Sched.aWeek[E_BA_Weekday.eFriday,1].stTime.nMinute		:= 0;
Sched.aWeek[E_BA_Weekday.eFriday,1].stTime.nSecond		:= 0;
Sched.aWeek[E_BA_Weekday.eFriday,2].eState				:= E_BA_SchedEntryState.eValue;
Sched.aWeek[E_BA_Weekday.eFriday,2].uValue.udiVal		:= E_BA_OnOff.eOff;
Sched.aWeek[E_BA_Weekday.eFriday,2].stTime.nHour		:= 5;
Sched.aWeek[E_BA_Weekday.eFriday,2].stTime.nMinute		:= 0;
Sched.aWeek[E_BA_Weekday.eFriday,2].stTime.nSecond		:= 0;
Sched.aWeek[E_BA_Weekday.eFriday,3].eState				:= E_BA_SchedEntryState.eValue;
Sched.aWeek[E_BA_Weekday.eFriday,3].uValue.udiVal		:= E_BA_OnOff.eOff;
Sched.aWeek[E_BA_Weekday.eFriday,3].stTime.nHour		:= 0;
Sched.aWeek[E_BA_Weekday.eFriday,3].stTime.nMinute		:= 0;
Sched.aWeek[E_BA_Weekday.eFriday,3].stTime.nSecond		:= 0;
Sched.bWriteException									:= FALSE;
END_METHOD

END_FUNCTION_BLOCK

// ---- Templates/POUs/Trade/AutomationControl/ControlCabinet/FB_BA_ControlCabinetBasicExt.TcPOU
{region '#Template'}
	{attribute 'Version' := '5.0.0.0'}
	{attribute 'Tags' := '"LCID": "1031", "Text": "General, Cabinet, Control cabinet, Acknowledgement"'}
	{attribute 'Tags' := '"LCID": "1033", "Text": "General, Cabinet, Control cabinet, Acknowledgement"'}
	{attribute 'Using' := '"Type": "Template", "URI": "BA2_Param"'}
	{attribute 'Using' := '"Type": "Template", "URI": "EC_ID"'}
	{attribute 'Description' := '"LCID": "1031", "Text": "Schaltschrank Quittierung"'}
	{attribute 'Description' := '"LCID": "1033", "Text": "Control cabinet acknowledgement"'}
{endregion}
FUNCTION_BLOCK FB_BA_ControlCabinetBasicExt EXTENDS FB_BA_View
VAR_INPUT
END_VAR
VAR_INPUT CONSTANT
	LampFault				: FB_BA_ActuatorCmd;		
	AckButton				: FB_BA_CombinationBI_BV;													
	EventObserver			: FB_BA_EventObserver;
END_VAR
VAR				
	bHasEvents				: BOOL;
	bHasUnackEvent			: BOOL;
	bTrigRstSwi				: BOOL;
	bTrigRstButton			: BOOL;	
END_VAR
VAR // added by the converter: edge detectors and wires of the graphical bodies
    _s1 : ST_BA_Binary;
END_VAR

SUPER^(); // FB_BA_View
AckButton(); // FB_BA_CombinationBI_BV
bTrigRstSwi := AckButton.bTrigBI_PrVal;
bTrigRstButton := AckButton.bTrigBV_PrVal;
EventObserver(bAck := bTrigRstSwi OR bTrigRstButton); // FB_BA_EventObserver
bHasEvents := EventObserver.bHasEvents;
bHasUnackEvent := EventObserver.bHasUnackEvents;
// compose _s1 : ST_BA_Binary
_s1.bEnPgm := bHasEvents;
_s1.bValPgm := SEL(bHasUnackEvent, TRUE, BA2_Param.bBlink);
LampFault(stCmd := _s1); // FB_BA_ActuatorCmd

METHOD FB_init : BOOL
VAR_INPUT
	bInitRetains : BOOL; // if TRUE, the retain variables are initialized (warm start / cold start)
	bInCopyCode : BOOL;  // if TRUE, the instance afterwards gets moved into the copy code (online change)
END_VAR
LampFault.iParent							:= THIS^;
LampFault.iLabel							:= LblCtl_EventIndicationLamp;
LampFault.eDPADMode							:= E_BA_DPADMode.eInclude;	
LampFault.Cmd.iLabel						:= LblFun_SwitchingCommand;		
LampFault.Cmd.ePolarity						:= E_BA_Polarity.eNormal;
LampFault.Cmd.sActiveText 					:= txtEvent_On;
LampFault.Cmd.sInactiveText 				:= txtEvent_Off;
LampFault.Cmd.nEventClassID					:= EC_ID.NC40;
LampFault.Cmd.aEventTransitionText[1]		:= txtEvent_Disturb;
LampFault.Cmd.aEventTransitionText[2]		:= txtEvent_None;
LampFault.Cmd.aEventTransitionText[3]		:= txtEvent_Normal;
LampFault.Cmd.bEventDetectionEnable			:= FALSE;
LampFault.Cmd.eEnPlantLock					:= E_BA_LockPriority.eNoLock;	

AckButton.iParent							:= THIS^;
AckButton.iLabel							:= LblCtl_Acknowledge;				
AckButton.eDPADMode							:= E_BA_DPADMode.eInclude;
AckButton.Input.iLabel						:= LblCtl_ButtonLocalAcknowledgement;																										
AckButton.Input.ePolarity					:= E_BA_Polarity.eNormal;
AckButton.Input.bEventDetectionEnable		:= FALSE;
AckButton.Value.eToggleMode 				:= E_BA_ToggleMode.ePushButton;					

EventObserver.Parent						:= XBA_Globals.Top;
END_METHOD

END_FUNCTION_BLOCK

// ---- Templates/POUs/Trade/AutomationControl/Device/BACnetSettings/FB_BACnet_RcpList.TcPOU
{region '#Template'}
	{attribute 'Version' := '5.0.0.0'}
	{attribute 'Tags' := '"LCID": "1031", "Text": "Automatisierungssteuerung, Gerät, Einstellungen, Projekt, Parameter"'}
	{attribute 'Tags' := '"LCID": "1033", "Text": "Automation control, Device, Settings, Project, Parameter"'}
	{attribute 'Description' := '"LCID": "1031", "Text": "Empfängerliste der Ereignisklassenobjekte / Meldungsklassenobjekte"'}
	{attribute 'Description' := '"LCID": "1033", "Text": "Recipient list of event class objects / notification class"'}
{endregion}

// Exemple illustrates how to write the (BACnet) recipient list to a 'FB_BA_EC' object.
FUNCTION_BLOCK FB_BACnet_RcpList  
VAR
	bWrite				: BOOL ;
	
	// Recipient list to write (to all event classes):
	aRecipientList		: T_BACnet_RecipientList := [(
							nProcessId					:= 10000,
							stValidDays					:= F_BACnet_ValidDays(TRUE, TRUE, TRUE, TRUE, TRUE, TRUE, TRUE),
							stFromTime					:= F_BA_ToSTTime(T#0H),
							stToTime					:= F_BA_ToSTTime(T#23H59M59S),
							bIssueConfirmed				:= FALSE,
							stEventTransitions			:= F_BACnet_EventTransitionBits(TRUE, TRUE, TRUE),
							stRecipient					:= F_BACnet_DeviceRecipient(nDeviceInstance:=1445709)
						),(
							nProcessId					:= 30100,
							stValidDays					:= F_BACnet_ValidDays(TRUE, TRUE, TRUE, TRUE, TRUE, FALSE, FALSE),
							stFromTime					:= F_BA_ToSTTime(T#0H),
							stToTime					:= F_BA_ToSTTime(T#23H59M59S),
							bIssueConfirmed				:= TRUE,
							stEventTransitions			:= F_BACnet_EventTransitionBits(TRUE, TRUE, TRUE),
							stRecipient					:= F_BACnet_EthernetRecipient(nIPAddress1:=192,168,10,200, nPort:=47808, nNetworkNr:=444)
						),(
							nProcessId					:= 40100,
							stValidDays					:= F_BACnet_ValidDays(TRUE, TRUE, TRUE, TRUE, FALSE, FALSE, FALSE),
							stFromTime					:= F_BA_ToSTTime(T#0H),
							stToTime					:= F_BA_ToSTTime(T#23H59M59S),
							bIssueConfirmed				:= TRUE,
							stEventTransitions			:= F_BACnet_EventTransitionBits(TRUE, TRUE, TRUE),
							stRecipient					:= F_BACnet_EthernetRecipient(nIPAddress1:=192,168,15,200, nPort:=47808, nNetworkNr:=555)
						)];
END_VAR
VAR
	bResult: BOOL;
	_iObj				: I_BA_Object;
	_fbBACnetObj		: POINTER TO FB_BACnet_BaseObject;
	_hRes				: HRESULT;
END_VAR

IF (XBA_Globals.Top.ProjectState = E_BA_ProjectState.eFirstOpCycle) THEN
	bWrite := TRUE;
END_IF


IF (bWrite) THEN
	bWrite := FALSE;
	// Iterate over all event class objects:
	_iObj := 0;
	WHILE (F_BA_IterateObjectIndex(_iObj, E_BA_ObjectType.eEventClass)) DO
		// Receive internal BACnet object from BA object:
		IF (NOT _iObj.GetBACnetObject(fbObject=>_fbBACnetObj)) THEN
			_iObj.LogMsg.Show(ADSLOG_MSGTYPE_ERROR, 'RL09', 'Failed to receive internal BACnet object!', TRUE);
		ELSE
			// Write recipient list:
			_hRes := _fbBACnetObj^.WritePropertyRecipientList(aRecipientList);
			IF (FAILED(_hRes)) THEN
				; // Do some error handling (An error message has already been logged here).
			END_IF
		END_IF
	END_WHILE
END_IF

END_FUNCTION_BLOCK

// ---- Templates/POUs/Trade/AutomationControl/EventClasses/FB_BA_EvtGroups.TcPOU
{region '#Template'}
	{attribute 'Version' := '5.0.0.0'}
	{attribute 'Tags' := '"LCID": "1031", "Text": "General, Cabinet, Control cabinet, Event groups, Categories, Notification classes, Event classes"'}
	{attribute 'Tags' := '"LCID": "1033", "Text": "General, Cabinet, Control cabinet, Event groups, Categories, Notification classes, Event classes"'}
	{attribute 'Using' := '"Type": "Template", "URI": "EC_ID"'}
	{attribute 'Description' := '"LCID": "1031", "Text": "Ereignisgruppen, Kategorien"'}
	{attribute 'Description' := '"LCID": "1033", "Text": "Event groups, categories"'}
{endregion}
FUNCTION_BLOCK FB_BA_EvtGroups EXTENDS FB_BA_View
VAR_INPUT CONSTANT
	LifeSafety						: FB_BA_EvtCategory;
	SafetyMsg						: FB_BA_EvtCategory;
	AlarmMsg						: FB_BA_EvtCategory;
	FaultMsg						: FB_BA_EvtCategory;
	MaintenanceMsg01				: FB_BA_EvtCategory;
	MaintenanceMsg02				: FB_BA_EvtCategory;
	SystemMsg						: FB_BA_EvtCategory;
	ManualOp						: FB_BA_EvtCategory;
	OtherMsg						: FB_BA_EvtCategory;
END_VAR

